	bArm1HorzULD1Unhook_00 AT %MX20356.0 : BOOL;
	bArm1HorzULD1Unhook_01 AT %MX20356.1 : BOOL;
	bArm1HorzULD1Unhook_02 AT %MX20356.2 : BOOL;
	bArm1HorzULD1Unhook_03 AT %MX20356.3 : BOOL;
	bArm1HorzULD1Unhook_04 AT %MX20356.4 : BOOL;
	bArm1HorzULD1Unhook_05 AT %MX20356.5 : BOOL;
	bArm1HorzULD1Unhook_06 AT %MX20356.6 : BOOL;
	bArm1HorzULD1Unhook_07 AT %MX20356.7 : BOOL;
	bArm1HorzULD1Unhook_08 AT %MX20356.8 : BOOL;
	bArm1HorzULD1Unhook_09 AT %MX20356.9 : BOOL;
	bArm1HorzULD1Unhook_10 AT %MX20356.10 : BOOL;
	bArm1HorzULD1Unhook_11 AT %MX20356.11 : BOOL;
	bArm1HorzULD1Unhook_12 AT %MX20356.12 : BOOL;
	bArm1HorzULD1Unhook_13 AT %MX20356.13 : BOOL;
	bArm1HorzULD1Unhook_14 AT %MX20356.14 : BOOL;
	bArm1HorzULD1Unhook_15 AT %MX20356.15 : BOOL;
	bArm1HorzULD1Unhook_16 AT %MX20356.16 : BOOL;
	bArm1HorzULD1Unhook_17 AT %MX20356.17 : BOOL;
	bArm1HorzULD1Unhook_18 AT %MX20356.18 : BOOL;
	bArm1HorzULD1Unhook_19 AT %MX20356.19 : BOOL;
	bArm1HorzULD1Unhook_20 AT %MX20356.20 : BOOL;
	bArm1HorzULD1Unhook_21 AT %MX20356.21 : BOOL;
	bArm1HorzULD1Unhook_22 AT %MX20356.22 : BOOL;
	bArm1HorzULD1Unhook_23 AT %MX20356.23 : BOOL;
	bArm1HorzULD1Unhook_24 AT %MX20356.24 : BOOL;
	bArm1HorzULD1Unhook_25 AT %MX20356.25 : BOOL;
	bArm1HorzULD1Unhook_26 AT %MX20356.26 : BOOL;
	bArm1HorzULD1Unhook_27 AT %MX20356.27 : BOOL;
	bArm1HorzULD1Unhook_28 AT %MX20356.28 : BOOL;
	bArm1HorzULD1Unhook_29 AT %MX20356.29 : BOOL;
	bArm1HorzULD1Unhook_30 AT %MX20356.30 : BOOL;
	bArm1HorzULD1Unhook_31 AT %MX20356.31 : BOOL;

	bArm1HorzStn1Unhook_00 AT %MX20304.0 : BOOL;
	bArm1HorzStn1Unhook_01 AT %MX20304.1 : BOOL;
	bArm1HorzStn1Unhook_02 AT %MX20304.2 : BOOL;
	bArm1HorzStn1Unhook_03 AT %MX20304.3 : BOOL;
	bArm1HorzStn1Unhook_04 AT %MX20304.4 : BOOL;
	bArm1HorzStn1Unhook_05 AT %MX20304.5 : BOOL;
	bArm1HorzStn1Unhook_06 AT %MX20304.6 : BOOL;
	bArm1HorzStn1Unhook_07 AT %MX20304.7 : BOOL;
	bArm1HorzStn1Unhook_08 AT %MX20304.8 : BOOL;
	bArm1HorzStn1Unhook_09 AT %MX20304.9 : BOOL;
	bArm1HorzStn1Unhook_10 AT %MX20304.10 : BOOL;
	bArm1HorzStn1Unhook_11 AT %MX20304.11 : BOOL;
	bArm1HorzStn1Unhook_12 AT %MX20304.12 : BOOL;
	bArm1HorzStn1Unhook_13 AT %MX20304.13 : BOOL;
	bArm1HorzStn1Unhook_14 AT %MX20304.14 : BOOL;
	bArm1HorzStn1Unhook_15 AT %MX20304.15 : BOOL;
	bArm1HorzStn1Unhook_16 AT %MX20304.16 : BOOL;
	bArm1HorzStn1Unhook_17 AT %MX20304.17 : BOOL;
	bArm1HorzStn1Unhook_18 AT %MX20304.18 : BOOL;
	bArm1HorzStn1Unhook_19 AT %MX20304.19 : BOOL;
	bArm1HorzStn1Unhook_20 AT %MX20304.20 : BOOL;
	bArm1HorzStn1Unhook_21 AT %MX20304.21 : BOOL;
	bArm1HorzStn1Unhook_22 AT %MX20304.22 : BOOL;
	bArm1HorzStn1Unhook_23 AT %MX20304.23 : BOOL;
	bArm1HorzStn1Unhook_24 AT %MX20304.24 : BOOL;
	bArm1HorzStn1Unhook_25 AT %MX20304.25 : BOOL;
	bArm1HorzStn1Unhook_26 AT %MX20304.26 : BOOL;
	bArm1HorzStn1Unhook_27 AT %MX20304.27 : BOOL;
	bArm1HorzStn1Unhook_28 AT %MX20304.28 : BOOL;
	bArm1HorzStn1Unhook_29 AT %MX20304.29 : BOOL;
	bArm1HorzStn1Unhook_30 AT %MX20304.30 : BOOL;
	bArm1HorzStn1Unhook_31 AT %MX20304.31 : BOOL;

	bArm1HorzStn2Unhook_00 AT %MX20308.0 : BOOL;
	bArm1HorzStn2Unhook_01 AT %MX20308.1 : BOOL;
	bArm1HorzStn2Unhook_02 AT %MX20308.2 : BOOL;
	bArm1HorzStn2Unhook_03 AT %MX20308.3 : BOOL;
	bArm1HorzStn2Unhook_04 AT %MX20308.4 : BOOL;
	bArm1HorzStn2Unhook_05 AT %MX20308.5 : BOOL;
	bArm1HorzStn2Unhook_06 AT %MX20308.6 : BOOL;
	bArm1HorzStn2Unhook_07 AT %MX20308.7 : BOOL;
	bArm1HorzStn2Unhook_08 AT %MX20308.8 : BOOL;
	bArm1HorzStn2Unhook_09 AT %MX20308.9 : BOOL;
	bArm1HorzStn2Unhook_10 AT %MX20308.10 : BOOL;
	bArm1HorzStn2Unhook_11 AT %MX20308.11 : BOOL;
	bArm1HorzStn2Unhook_12 AT %MX20308.12 : BOOL;
	bArm1HorzStn2Unhook_13 AT %MX20308.13 : BOOL;
	bArm1HorzStn2Unhook_14 AT %MX20308.14 : BOOL;
	bArm1HorzStn2Unhook_15 AT %MX20308.15 : BOOL;
	bArm1HorzStn2Unhook_16 AT %MX20308.16 : BOOL;
	bArm1HorzStn2Unhook_17 AT %MX20308.17 : BOOL;
	bArm1HorzStn2Unhook_18 AT %MX20308.18 : BOOL;
	bArm1HorzStn2Unhook_19 AT %MX20308.19 : BOOL;
	bArm1HorzStn2Unhook_20 AT %MX20308.20 : BOOL;
	bArm1HorzStn2Unhook_21 AT %MX20308.21 : BOOL;
	bArm1HorzStn2Unhook_22 AT %MX20308.22 : BOOL;
	bArm1HorzStn2Unhook_23 AT %MX20308.23 : BOOL;
	bArm1HorzStn2Unhook_24 AT %MX20308.24 : BOOL;
	bArm1HorzStn2Unhook_25 AT %MX20308.25 : BOOL;
	bArm1HorzStn2Unhook_26 AT %MX20308.26 : BOOL;
	bArm1HorzStn2Unhook_27 AT %MX20308.27 : BOOL;
	bArm1HorzStn2Unhook_28 AT %MX20308.28 : BOOL;
	bArm1HorzStn2Unhook_29 AT %MX20308.29 : BOOL;
	bArm1HorzStn2Unhook_30 AT %MX20308.30 : BOOL;
	bArm1HorzStn2Unhook_31 AT %MX20308.31 : BOOL;

	bArm1HorzStn3Unhook_00 AT %MX20312.0 : BOOL;
	bArm1HorzStn3Unhook_01 AT %MX20312.1 : BOOL;
	bArm1HorzStn3Unhook_02 AT %MX20312.2 : BOOL;
	bArm1HorzStn3Unhook_03 AT %MX20312.3 : BOOL;
	bArm1HorzStn3Unhook_04 AT %MX20312.4 : BOOL;
	bArm1HorzStn3Unhook_05 AT %MX20312.5 : BOOL;
	bArm1HorzStn3Unhook_06 AT %MX20312.6 : BOOL;
	bArm1HorzStn3Unhook_07 AT %MX20312.7 : BOOL;
	bArm1HorzStn3Unhook_08 AT %MX20312.8 : BOOL;
	bArm1HorzStn3Unhook_09 AT %MX20312.9 : BOOL;
	bArm1HorzStn3Unhook_10 AT %MX20312.10 : BOOL;
	bArm1HorzStn3Unhook_11 AT %MX20312.11 : BOOL;
	bArm1HorzStn3Unhook_12 AT %MX20312.12 : BOOL;
	bArm1HorzStn3Unhook_13 AT %MX20312.13 : BOOL;
	bArm1HorzStn3Unhook_14 AT %MX20312.14 : BOOL;
	bArm1HorzStn3Unhook_15 AT %MX20312.15 : BOOL;
	bArm1HorzStn3Unhook_16 AT %MX20312.16 : BOOL;
	bArm1HorzStn3Unhook_17 AT %MX20312.17 : BOOL;
	bArm1HorzStn3Unhook_18 AT %MX20312.18 : BOOL;
	bArm1HorzStn3Unhook_19 AT %MX20312.19 : BOOL;
	bArm1HorzStn3Unhook_20 AT %MX20312.20 : BOOL;
	bArm1HorzStn3Unhook_21 AT %MX20312.21 : BOOL;
	bArm1HorzStn3Unhook_22 AT %MX20312.22 : BOOL;
	bArm1HorzStn3Unhook_23 AT %MX20312.23 : BOOL;
	bArm1HorzStn3Unhook_24 AT %MX20312.24 : BOOL;
	bArm1HorzStn3Unhook_25 AT %MX20312.25 : BOOL;
	bArm1HorzStn3Unhook_26 AT %MX20312.26 : BOOL;
	bArm1HorzStn3Unhook_27 AT %MX20312.27 : BOOL;
	bArm1HorzStn3Unhook_28 AT %MX20312.28 : BOOL;
	bArm1HorzStn3Unhook_29 AT %MX20312.29 : BOOL;
	bArm1HorzStn3Unhook_30 AT %MX20312.30 : BOOL;
	bArm1HorzStn3Unhook_31 AT %MX20312.31 : BOOL;

	bArm1HorzStn4Unhook_00 AT %MX20316.0 : BOOL;
	bArm1HorzStn4Unhook_01 AT %MX20316.1 : BOOL;
	bArm1HorzStn4Unhook_02 AT %MX20316.2 : BOOL;
	bArm1HorzStn4Unhook_03 AT %MX20316.3 : BOOL;
	bArm1HorzStn4Unhook_04 AT %MX20316.4 : BOOL;
	bArm1HorzStn4Unhook_05 AT %MX20316.5 : BOOL;
	bArm1HorzStn4Unhook_06 AT %MX20316.6 : BOOL;
	bArm1HorzStn4Unhook_07 AT %MX20316.7 : BOOL;
	bArm1HorzStn4Unhook_08 AT %MX20316.8 : BOOL;
	bArm1HorzStn4Unhook_09 AT %MX20316.9 : BOOL;
	bArm1HorzStn4Unhook_10 AT %MX20316.10 : BOOL;
	bArm1HorzStn4Unhook_11 AT %MX20316.11 : BOOL;
	bArm1HorzStn4Unhook_12 AT %MX20316.12 : BOOL;
	bArm1HorzStn4Unhook_13 AT %MX20316.13 : BOOL;
	bArm1HorzStn4Unhook_14 AT %MX20316.14 : BOOL;
	bArm1HorzStn4Unhook_15 AT %MX20316.15 : BOOL;
	bArm1HorzStn4Unhook_16 AT %MX20316.16 : BOOL;
	bArm1HorzStn4Unhook_17 AT %MX20316.17 : BOOL;
	bArm1HorzStn4Unhook_18 AT %MX20316.18 : BOOL;
	bArm1HorzStn4Unhook_19 AT %MX20316.19 : BOOL;
	bArm1HorzStn4Unhook_20 AT %MX20316.20 : BOOL;
	bArm1HorzStn4Unhook_21 AT %MX20316.21 : BOOL;
	bArm1HorzStn4Unhook_22 AT %MX20316.22 : BOOL;
	bArm1HorzStn4Unhook_23 AT %MX20316.23 : BOOL;
	bArm1HorzStn4Unhook_24 AT %MX20316.24 : BOOL;
	bArm1HorzStn4Unhook_25 AT %MX20316.25 : BOOL;
	bArm1HorzStn4Unhook_26 AT %MX20316.26 : BOOL;
	bArm1HorzStn4Unhook_27 AT %MX20316.27 : BOOL;
	bArm1HorzStn4Unhook_28 AT %MX20316.28 : BOOL;
	bArm1HorzStn4Unhook_29 AT %MX20316.29 : BOOL;
	bArm1HorzStn4Unhook_30 AT %MX20316.30 : BOOL;
	bArm1HorzStn4Unhook_31 AT %MX20316.31 : BOOL;

	bArm1HorzStn5Unhook_00 AT %MX20320.0 : BOOL;
	bArm1HorzStn5Unhook_01 AT %MX20320.1 : BOOL;
	bArm1HorzStn5Unhook_02 AT %MX20320.2 : BOOL;
	bArm1HorzStn5Unhook_03 AT %MX20320.3 : BOOL;
	bArm1HorzStn5Unhook_04 AT %MX20320.4 : BOOL;
	bArm1HorzStn5Unhook_05 AT %MX20320.5 : BOOL;
	bArm1HorzStn5Unhook_06 AT %MX20320.6 : BOOL;
	bArm1HorzStn5Unhook_07 AT %MX20320.7 : BOOL;
	bArm1HorzStn5Unhook_08 AT %MX20320.8 : BOOL;
	bArm1HorzStn5Unhook_09 AT %MX20320.9 : BOOL;
	bArm1HorzStn5Unhook_10 AT %MX20320.10 : BOOL;
	bArm1HorzStn5Unhook_11 AT %MX20320.11 : BOOL;
	bArm1HorzStn5Unhook_12 AT %MX20320.12 : BOOL;
	bArm1HorzStn5Unhook_13 AT %MX20320.13 : BOOL;
	bArm1HorzStn5Unhook_14 AT %MX20320.14 : BOOL;
	bArm1HorzStn5Unhook_15 AT %MX20320.15 : BOOL;
	bArm1HorzStn5Unhook_16 AT %MX20320.16 : BOOL;
	bArm1HorzStn5Unhook_17 AT %MX20320.17 : BOOL;
	bArm1HorzStn5Unhook_18 AT %MX20320.18 : BOOL;
	bArm1HorzStn5Unhook_19 AT %MX20320.19 : BOOL;
	bArm1HorzStn5Unhook_20 AT %MX20320.20 : BOOL;
	bArm1HorzStn5Unhook_21 AT %MX20320.21 : BOOL;
	bArm1HorzStn5Unhook_22 AT %MX20320.22 : BOOL;
	bArm1HorzStn5Unhook_23 AT %MX20320.23 : BOOL;
	bArm1HorzStn5Unhook_24 AT %MX20320.24 : BOOL;
	bArm1HorzStn5Unhook_25 AT %MX20320.25 : BOOL;
	bArm1HorzStn5Unhook_26 AT %MX20320.26 : BOOL;
	bArm1HorzStn5Unhook_27 AT %MX20320.27 : BOOL;
	bArm1HorzStn5Unhook_28 AT %MX20320.28 : BOOL;
	bArm1HorzStn5Unhook_29 AT %MX20320.29 : BOOL;
	bArm1HorzStn5Unhook_30 AT %MX20320.30 : BOOL;
	bArm1HorzStn5Unhook_31 AT %MX20320.31 : BOOL;

	bArm1HorzStn6Unhook_00 AT %MX20324.0 : BOOL;
	bArm1HorzStn6Unhook_01 AT %MX20324.1 : BOOL;
	bArm1HorzStn6Unhook_02 AT %MX20324.2 : BOOL;
	bArm1HorzStn6Unhook_03 AT %MX20324.3 : BOOL;
	bArm1HorzStn6Unhook_04 AT %MX20324.4 : BOOL;
	bArm1HorzStn6Unhook_05 AT %MX20324.5 : BOOL;
	bArm1HorzStn6Unhook_06 AT %MX20324.6 : BOOL;
	bArm1HorzStn6Unhook_07 AT %MX20324.7 : BOOL;
	bArm1HorzStn6Unhook_08 AT %MX20324.8 : BOOL;
	bArm1HorzStn6Unhook_09 AT %MX20324.9 : BOOL;
	bArm1HorzStn6Unhook_10 AT %MX20324.10 : BOOL;
	bArm1HorzStn6Unhook_11 AT %MX20324.11 : BOOL;
	bArm1HorzStn6Unhook_12 AT %MX20324.12 : BOOL;
	bArm1HorzStn6Unhook_13 AT %MX20324.13 : BOOL;
	bArm1HorzStn6Unhook_14 AT %MX20324.14 : BOOL;
	bArm1HorzStn6Unhook_15 AT %MX20324.15 : BOOL;
	bArm1HorzStn6Unhook_16 AT %MX20324.16 : BOOL;
	bArm1HorzStn6Unhook_17 AT %MX20324.17 : BOOL;
	bArm1HorzStn6Unhook_18 AT %MX20324.18 : BOOL;
	bArm1HorzStn6Unhook_19 AT %MX20324.19 : BOOL;
	bArm1HorzStn6Unhook_20 AT %MX20324.20 : BOOL;
	bArm1HorzStn6Unhook_21 AT %MX20324.21 : BOOL;
	bArm1HorzStn6Unhook_22 AT %MX20324.22 : BOOL;
	bArm1HorzStn6Unhook_23 AT %MX20324.23 : BOOL;
	bArm1HorzStn6Unhook_24 AT %MX20324.24 : BOOL;
	bArm1HorzStn6Unhook_25 AT %MX20324.25 : BOOL;
	bArm1HorzStn6Unhook_26 AT %MX20324.26 : BOOL;
	bArm1HorzStn6Unhook_27 AT %MX20324.27 : BOOL;
	bArm1HorzStn6Unhook_28 AT %MX20324.28 : BOOL;
	bArm1HorzStn6Unhook_29 AT %MX20324.29 : BOOL;
	bArm1HorzStn6Unhook_30 AT %MX20324.30 : BOOL;
	bArm1HorzStn6Unhook_31 AT %MX20324.31 : BOOL;

	bArm1HorzStn7Unhook_00 AT %MX20328.0 : BOOL;
	bArm1HorzStn7Unhook_01 AT %MX20328.1 : BOOL;
	bArm1HorzStn7Unhook_02 AT %MX20328.2 : BOOL;
	bArm1HorzStn7Unhook_03 AT %MX20328.3 : BOOL;
	bArm1HorzStn7Unhook_04 AT %MX20328.4 : BOOL;
	bArm1HorzStn7Unhook_05 AT %MX20328.5 : BOOL;
	bArm1HorzStn7Unhook_06 AT %MX20328.6 : BOOL;
	bArm1HorzStn7Unhook_07 AT %MX20328.7 : BOOL;
	bArm1HorzStn7Unhook_08 AT %MX20328.8 : BOOL;
	bArm1HorzStn7Unhook_09 AT %MX20328.9 : BOOL;
	bArm1HorzStn7Unhook_10 AT %MX20328.10 : BOOL;
	bArm1HorzStn7Unhook_11 AT %MX20328.11 : BOOL;
	bArm1HorzStn7Unhook_12 AT %MX20328.12 : BOOL;
	bArm1HorzStn7Unhook_13 AT %MX20328.13 : BOOL;
	bArm1HorzStn7Unhook_14 AT %MX20328.14 : BOOL;
	bArm1HorzStn7Unhook_15 AT %MX20328.15 : BOOL;
	bArm1HorzStn7Unhook_16 AT %MX20328.16 : BOOL;
	bArm1HorzStn7Unhook_17 AT %MX20328.17 : BOOL;
	bArm1HorzStn7Unhook_18 AT %MX20328.18 : BOOL;
	bArm1HorzStn7Unhook_19 AT %MX20328.19 : BOOL;
	bArm1HorzStn7Unhook_20 AT %MX20328.20 : BOOL;
	bArm1HorzStn7Unhook_21 AT %MX20328.21 : BOOL;
	bArm1HorzStn7Unhook_22 AT %MX20328.22 : BOOL;
	bArm1HorzStn7Unhook_23 AT %MX20328.23 : BOOL;
	bArm1HorzStn7Unhook_24 AT %MX20328.24 : BOOL;
	bArm1HorzStn7Unhook_25 AT %MX20328.25 : BOOL;
	bArm1HorzStn7Unhook_26 AT %MX20328.26 : BOOL;
	bArm1HorzStn7Unhook_27 AT %MX20328.27 : BOOL;
	bArm1HorzStn7Unhook_28 AT %MX20328.28 : BOOL;
	bArm1HorzStn7Unhook_29 AT %MX20328.29 : BOOL;
	bArm1HorzStn7Unhook_30 AT %MX20328.30 : BOOL;
	bArm1HorzStn7Unhook_31 AT %MX20328.31 : BOOL;

	bArm1HorzStn8Unhook_00 AT %MX20332.0 : BOOL;
	bArm1HorzStn8Unhook_01 AT %MX20332.1 : BOOL;
	bArm1HorzStn8Unhook_02 AT %MX20332.2 : BOOL;
	bArm1HorzStn8Unhook_03 AT %MX20332.3 : BOOL;
	bArm1HorzStn8Unhook_04 AT %MX20332.4 : BOOL;
	bArm1HorzStn8Unhook_05 AT %MX20332.5 : BOOL;
	bArm1HorzStn8Unhook_06 AT %MX20332.6 : BOOL;
	bArm1HorzStn8Unhook_07 AT %MX20332.7 : BOOL;
	bArm1HorzStn8Unhook_08 AT %MX20332.8 : BOOL;
	bArm1HorzStn8Unhook_09 AT %MX20332.9 : BOOL;
	bArm1HorzStn8Unhook_10 AT %MX20332.10 : BOOL;
	bArm1HorzStn8Unhook_11 AT %MX20332.11 : BOOL;
	bArm1HorzStn8Unhook_12 AT %MX20332.12 : BOOL;
	bArm1HorzStn8Unhook_13 AT %MX20332.13 : BOOL;
	bArm1HorzStn8Unhook_14 AT %MX20332.14 : BOOL;
	bArm1HorzStn8Unhook_15 AT %MX20332.15 : BOOL;
	bArm1HorzStn8Unhook_16 AT %MX20332.16 : BOOL;
	bArm1HorzStn8Unhook_17 AT %MX20332.17 : BOOL;
	bArm1HorzStn8Unhook_18 AT %MX20332.18 : BOOL;
	bArm1HorzStn8Unhook_19 AT %MX20332.19 : BOOL;
	bArm1HorzStn8Unhook_20 AT %MX20332.20 : BOOL;
	bArm1HorzStn8Unhook_21 AT %MX20332.21 : BOOL;
	bArm1HorzStn8Unhook_22 AT %MX20332.22 : BOOL;
	bArm1HorzStn8Unhook_23 AT %MX20332.23 : BOOL;
	bArm1HorzStn8Unhook_24 AT %MX20332.24 : BOOL;
	bArm1HorzStn8Unhook_25 AT %MX20332.25 : BOOL;
	bArm1HorzStn8Unhook_26 AT %MX20332.26 : BOOL;
	bArm1HorzStn8Unhook_27 AT %MX20332.27 : BOOL;
	bArm1HorzStn8Unhook_28 AT %MX20332.28 : BOOL;
	bArm1HorzStn8Unhook_29 AT %MX20332.29 : BOOL;
	bArm1HorzStn8Unhook_30 AT %MX20332.30 : BOOL;
	bArm1HorzStn8Unhook_31 AT %MX20332.31 : BOOL;

	bArm1HorzStn9Unhook_00 AT %MX20336.0 : BOOL;
	bArm1HorzStn9Unhook_01 AT %MX20336.1 : BOOL;
	bArm1HorzStn9Unhook_02 AT %MX20336.2 : BOOL;
	bArm1HorzStn9Unhook_03 AT %MX20336.3 : BOOL;
	bArm1HorzStn9Unhook_04 AT %MX20336.4 : BOOL;
	bArm1HorzStn9Unhook_05 AT %MX20336.5 : BOOL;
	bArm1HorzStn9Unhook_06 AT %MX20336.6 : BOOL;
	bArm1HorzStn9Unhook_07 AT %MX20336.7 : BOOL;
	bArm1HorzStn9Unhook_08 AT %MX20336.8 : BOOL;
	bArm1HorzStn9Unhook_09 AT %MX20336.9 : BOOL;
	bArm1HorzStn9Unhook_10 AT %MX20336.10 : BOOL;
	bArm1HorzStn9Unhook_11 AT %MX20336.11 : BOOL;
	bArm1HorzStn9Unhook_12 AT %MX20336.12 : BOOL;
	bArm1HorzStn9Unhook_13 AT %MX20336.13 : BOOL;
	bArm1HorzStn9Unhook_14 AT %MX20336.14 : BOOL;
	bArm1HorzStn9Unhook_15 AT %MX20336.15 : BOOL;
	bArm1HorzStn9Unhook_16 AT %MX20336.16 : BOOL;
	bArm1HorzStn9Unhook_17 AT %MX20336.17 : BOOL;
	bArm1HorzStn9Unhook_18 AT %MX20336.18 : BOOL;
	bArm1HorzStn9Unhook_19 AT %MX20336.19 : BOOL;
	bArm1HorzStn9Unhook_20 AT %MX20336.20 : BOOL;
	bArm1HorzStn9Unhook_21 AT %MX20336.21 : BOOL;
	bArm1HorzStn9Unhook_22 AT %MX20336.22 : BOOL;
	bArm1HorzStn9Unhook_23 AT %MX20336.23 : BOOL;
	bArm1HorzStn9Unhook_24 AT %MX20336.24 : BOOL;
	bArm1HorzStn9Unhook_25 AT %MX20336.25 : BOOL;
	bArm1HorzStn9Unhook_26 AT %MX20336.26 : BOOL;
	bArm1HorzStn9Unhook_27 AT %MX20336.27 : BOOL;
	bArm1HorzStn9Unhook_28 AT %MX20336.28 : BOOL;
	bArm1HorzStn9Unhook_29 AT %MX20336.29 : BOOL;
	bArm1HorzStn9Unhook_30 AT %MX20336.30 : BOOL;
	bArm1HorzStn9Unhook_31 AT %MX20336.31 : BOOL;

	bArm1HorzStn10Unhook_00 AT %MX20340.0 : BOOL;
	bArm1HorzStn10Unhook_01 AT %MX20340.1 : BOOL;
	bArm1HorzStn10Unhook_02 AT %MX20340.2 : BOOL;
	bArm1HorzStn10Unhook_03 AT %MX20340.3 : BOOL;
	bArm1HorzStn10Unhook_04 AT %MX20340.4 : BOOL;
	bArm1HorzStn10Unhook_05 AT %MX20340.5 : BOOL;
	bArm1HorzStn10Unhook_06 AT %MX20340.6 : BOOL;
	bArm1HorzStn10Unhook_07 AT %MX20340.7 : BOOL;
	bArm1HorzStn10Unhook_08 AT %MX20340.8 : BOOL;
	bArm1HorzStn10Unhook_09 AT %MX20340.9 : BOOL;
	bArm1HorzStn10Unhook_10 AT %MX20340.10 : BOOL;
	bArm1HorzStn10Unhook_11 AT %MX20340.11 : BOOL;
	bArm1HorzStn10Unhook_12 AT %MX20340.12 : BOOL;
	bArm1HorzStn10Unhook_13 AT %MX20340.13 : BOOL;
	bArm1HorzStn10Unhook_14 AT %MX20340.14 : BOOL;
	bArm1HorzStn10Unhook_15 AT %MX20340.15 : BOOL;
	bArm1HorzStn10Unhook_16 AT %MX20340.16 : BOOL;
	bArm1HorzStn10Unhook_17 AT %MX20340.17 : BOOL;
	bArm1HorzStn10Unhook_18 AT %MX20340.18 : BOOL;
	bArm1HorzStn10Unhook_19 AT %MX20340.19 : BOOL;
	bArm1HorzStn10Unhook_20 AT %MX20340.20 : BOOL;
	bArm1HorzStn10Unhook_21 AT %MX20340.21 : BOOL;
	bArm1HorzStn10Unhook_22 AT %MX20340.22 : BOOL;
	bArm1HorzStn10Unhook_23 AT %MX20340.23 : BOOL;
	bArm1HorzStn10Unhook_24 AT %MX20340.24 : BOOL;
	bArm1HorzStn10Unhook_25 AT %MX20340.25 : BOOL;
	bArm1HorzStn10Unhook_26 AT %MX20340.26 : BOOL;
	bArm1HorzStn10Unhook_27 AT %MX20340.27 : BOOL;
	bArm1HorzStn10Unhook_28 AT %MX20340.28 : BOOL;
	bArm1HorzStn10Unhook_29 AT %MX20340.29 : BOOL;
	bArm1HorzStn10Unhook_30 AT %MX20340.30 : BOOL;
	bArm1HorzStn10Unhook_31 AT %MX20340.31 : BOOL;

	bArm1HorzStn11Unhook_00 AT %MX20344.0 : BOOL;
	bArm1HorzStn11Unhook_01 AT %MX20344.1 : BOOL;
	bArm1HorzStn11Unhook_02 AT %MX20344.2 : BOOL;
	bArm1HorzStn11Unhook_03 AT %MX20344.3 : BOOL;
	bArm1HorzStn11Unhook_04 AT %MX20344.4 : BOOL;
	bArm1HorzStn11Unhook_05 AT %MX20344.5 : BOOL;
	bArm1HorzStn11Unhook_06 AT %MX20344.6 : BOOL;
	bArm1HorzStn11Unhook_07 AT %MX20344.7 : BOOL;
	bArm1HorzStn11Unhook_08 AT %MX20344.8 : BOOL;
	bArm1HorzStn11Unhook_09 AT %MX20344.9 : BOOL;
	bArm1HorzStn11Unhook_10 AT %MX20344.10 : BOOL;
	bArm1HorzStn11Unhook_11 AT %MX20344.11 : BOOL;
	bArm1HorzStn11Unhook_12 AT %MX20344.12 : BOOL;
	bArm1HorzStn11Unhook_13 AT %MX20344.13 : BOOL;
	bArm1HorzStn11Unhook_14 AT %MX20344.14 : BOOL;
	bArm1HorzStn11Unhook_15 AT %MX20344.15 : BOOL;
	bArm1HorzStn11Unhook_16 AT %MX20344.16 : BOOL;
	bArm1HorzStn11Unhook_17 AT %MX20344.17 : BOOL;
	bArm1HorzStn11Unhook_18 AT %MX20344.18 : BOOL;
	bArm1HorzStn11Unhook_19 AT %MX20344.19 : BOOL;
	bArm1HorzStn11Unhook_20 AT %MX20344.20 : BOOL;
	bArm1HorzStn11Unhook_21 AT %MX20344.21 : BOOL;
	bArm1HorzStn11Unhook_22 AT %MX20344.22 : BOOL;
	bArm1HorzStn11Unhook_23 AT %MX20344.23 : BOOL;
	bArm1HorzStn11Unhook_24 AT %MX20344.24 : BOOL;
	bArm1HorzStn11Unhook_25 AT %MX20344.25 : BOOL;
	bArm1HorzStn11Unhook_26 AT %MX20344.26 : BOOL;
	bArm1HorzStn11Unhook_27 AT %MX20344.27 : BOOL;
	bArm1HorzStn11Unhook_28 AT %MX20344.28 : BOOL;
	bArm1HorzStn11Unhook_29 AT %MX20344.29 : BOOL;
	bArm1HorzStn11Unhook_30 AT %MX20344.30 : BOOL;
	bArm1HorzStn11Unhook_31 AT %MX20344.31 : BOOL;

	bArm1HorzStn12Unhook_00 AT %MX20348.0 : BOOL;
	bArm1HorzStn12Unhook_01 AT %MX20348.1 : BOOL;
	bArm1HorzStn12Unhook_02 AT %MX20348.2 : BOOL;
	bArm1HorzStn12Unhook_03 AT %MX20348.3 : BOOL;
	bArm1HorzStn12Unhook_04 AT %MX20348.4 : BOOL;
	bArm1HorzStn12Unhook_05 AT %MX20348.5 : BOOL;
	bArm1HorzStn12Unhook_06 AT %MX20348.6 : BOOL;
	bArm1HorzStn12Unhook_07 AT %MX20348.7 : BOOL;
	bArm1HorzStn12Unhook_08 AT %MX20348.8 : BOOL;
	bArm1HorzStn12Unhook_09 AT %MX20348.9 : BOOL;
	bArm1HorzStn12Unhook_10 AT %MX20348.10 : BOOL;
	bArm1HorzStn12Unhook_11 AT %MX20348.11 : BOOL;
	bArm1HorzStn12Unhook_12 AT %MX20348.12 : BOOL;
	bArm1HorzStn12Unhook_13 AT %MX20348.13 : BOOL;
	bArm1HorzStn12Unhook_14 AT %MX20348.14 : BOOL;
	bArm1HorzStn12Unhook_15 AT %MX20348.15 : BOOL;
	bArm1HorzStn12Unhook_16 AT %MX20348.16 : BOOL;
	bArm1HorzStn12Unhook_17 AT %MX20348.17 : BOOL;
	bArm1HorzStn12Unhook_18 AT %MX20348.18 : BOOL;
	bArm1HorzStn12Unhook_19 AT %MX20348.19 : BOOL;
	bArm1HorzStn12Unhook_20 AT %MX20348.20 : BOOL;
	bArm1HorzStn12Unhook_21 AT %MX20348.21 : BOOL;
	bArm1HorzStn12Unhook_22 AT %MX20348.22 : BOOL;
	bArm1HorzStn12Unhook_23 AT %MX20348.23 : BOOL;
	bArm1HorzStn12Unhook_24 AT %MX20348.24 : BOOL;
	bArm1HorzStn12Unhook_25 AT %MX20348.25 : BOOL;
	bArm1HorzStn12Unhook_26 AT %MX20348.26 : BOOL;
	bArm1HorzStn12Unhook_27 AT %MX20348.27 : BOOL;
	bArm1HorzStn12Unhook_28 AT %MX20348.28 : BOOL;
	bArm1HorzStn12Unhook_29 AT %MX20348.29 : BOOL;
	bArm1HorzStn12Unhook_30 AT %MX20348.30 : BOOL;
	bArm1HorzStn12Unhook_31 AT %MX20348.31 : BOOL;


(* xxxxxxxxxxxxxxxxxxxxxxxxxxxxxxxxxxxxxxx Vert xxxxxxxxxxxxxxxxxxxxxxxxxxxxxxxxxxxxxxx*)
(*========= Up BOOL LINK with %MX25000-MX25099 =========*)

	bArm1VertLD1Up_00 AT %MX25052.0 : BOOL;
	bArm1VertLD1Up_01 AT %MX25052.1 : BOOL;
	bArm1VertLD1Up_02 AT %MX25052.2 : BOOL;
	bArm1VertLD1Up_03 AT %MX25052.3 : BOOL;
	bArm1VertLD1Up_04 AT %MX25052.4 : BOOL;
	bArm1VertLD1Up_05 AT %MX25052.5 : BOOL;
	bArm1VertLD1Up_06 AT %MX25052.6 : BOOL;
	bArm1VertLD1Up_07 AT %MX25052.7 : BOOL;
	bArm1VertLD1Up_08 AT %MX25052.8 : BOOL;
	bArm1VertLD1Up_09 AT %MX25052.9 : BOOL;
	bArm1VertLD1Up_10 AT %MX25052.10 : BOOL;
	bArm1VertLD1Up_11 AT %MX25052.11 : BOOL;
	bArm1VertLD1Up_12 AT %MX25052.12 : BOOL;
	bArm1VertLD1Up_13 AT %MX25052.13 : BOOL;
	bArm1VertLD1Up_14 AT %MX25052.14 : BOOL;
	bArm1VertLD1Up_15 AT %MX25052.15 : BOOL;
	bArm1VertLD1Up_16 AT %MX25052.16 : BOOL;
	bArm1VertLD1Up_17 AT %MX25052.17 : BOOL;
	bArm1VertLD1Up_18 AT %MX25052.18 : BOOL;
	bArm1VertLD1Up_19 AT %MX25052.19 : BOOL;
	bArm1VertLD1Up_20 AT %MX25052.20 : BOOL;
	bArm1VertLD1Up_21 AT %MX25052.21 : BOOL;
	bArm1VertLD1Up_22 AT %MX25052.22 : BOOL;
	bArm1VertLD1Up_23 AT %MX25052.23 : BOOL;
	bArm1VertLD1Up_24 AT %MX25052.24 : BOOL;
	bArm1VertLD1Up_25 AT %MX25052.25 : BOOL;
	bArm1VertLD1Up_26 AT %MX25052.26 : BOOL;
	bArm1VertLD1Up_27 AT %MX25052.27 : BOOL;
	bArm1VertLD1Up_28 AT %MX25052.28 : BOOL;
	bArm1VertLD1Up_29 AT %MX25052.29 : BOOL;
	bArm1VertLD1Up_30 AT %MX25052.30 : BOOL;
	bArm1VertLD1Up_31 AT %MX25052.31 : BOOL;

	bArm1VertULD1Up_00 AT %MX25056.0 : BOOL;
	bArm1VertULD1Up_01 AT %MX25056.1 : BOOL;
	bArm1VertULD1Up_02 AT %MX25056.2 : BOOL;
	bArm1VertULD1Up_03 AT %MX25056.3 : BOOL;
	bArm1VertULD1Up_04 AT %MX25056.4 : BOOL;
	bArm1VertULD1Up_05 AT %MX25056.5 : BOOL;
	bArm1VertULD1Up_06 AT %MX25056.6 : BOOL;
	bArm1VertULD1Up_07 AT %MX25056.7 : BOOL;
	bArm1VertULD1Up_08 AT %MX25056.8 : BOOL;
	bArm1VertULD1Up_09 AT %MX25056.9 : BOOL;
	bArm1VertULD1Up_10 AT %MX25056.10 : BOOL;
	bArm1VertULD1Up_11 AT %MX25056.11 : BOOL;
	bArm1VertULD1Up_12 AT %MX25056.12 : BOOL;
	bArm1VertULD1Up_13 AT %MX25056.13 : BOOL;
	bArm1VertULD1Up_14 AT %MX25056.14 : BOOL;
	bArm1VertULD1Up_15 AT %MX25056.15 : BOOL;
	bArm1VertULD1Up_16 AT %MX25056.16 : BOOL;
	bArm1VertULD1Up_17 AT %MX25056.17 : BOOL;
	bArm1VertULD1Up_18 AT %MX25056.18 : BOOL;
	bArm1VertULD1Up_19 AT %MX25056.19 : BOOL;
	bArm1VertULD1Up_20 AT %MX25056.20 : BOOL;
	bArm1VertULD1Up_21 AT %MX25056.21 : BOOL;
	bArm1VertULD1Up_22 AT %MX25056.22 : BOOL;
	bArm1VertULD1Up_23 AT %MX25056.23 : BOOL;
	bArm1VertULD1Up_24 AT %MX25056.24 : BOOL;
	bArm1VertULD1Up_25 AT %MX25056.25 : BOOL;
	bArm1VertULD1Up_26 AT %MX25056.26 : BOOL;
	bArm1VertULD1Up_27 AT %MX25056.27 : BOOL;
	bArm1VertULD1Up_28 AT %MX25056.28 : BOOL;
	bArm1VertULD1Up_29 AT %MX25056.29 : BOOL;
	bArm1VertULD1Up_30 AT %MX25056.30 : BOOL;
	bArm1VertULD1Up_31 AT %MX25056.31 : BOOL;

	bArm1VertStn1Up_00 AT %MX25004.0 : BOOL;
	bArm1VertStn1Up_01 AT %MX25004.1 : BOOL;
	bArm1VertStn1Up_02 AT %MX25004.2 : BOOL;
	bArm1VertStn1Up_03 AT %MX25004.3 : BOOL;
	bArm1VertStn1Up_04 AT %MX25004.4 : BOOL;
	bArm1VertStn1Up_05 AT %MX25004.5 : BOOL;
	bArm1VertStn1Up_06 AT %MX25004.6 : BOOL;
	bArm1VertStn1Up_07 AT %MX25004.7 : BOOL;
	bArm1VertStn1Up_08 AT %MX25004.8 : BOOL;
	bArm1VertStn1Up_09 AT %MX25004.9 : BOOL;
	bArm1VertStn1Up_10 AT %MX25004.10 : BOOL;
	bArm1VertStn1Up_11 AT %MX25004.11 : BOOL;
	bArm1VertStn1Up_12 AT %MX25004.12 : BOOL;
	bArm1VertStn1Up_13 AT %MX25004.13 : BOOL;
	bArm1VertStn1Up_14 AT %MX25004.14 : BOOL;
	bArm1VertStn1Up_15 AT %MX25004.15 : BOOL;
	bArm1VertStn1Up_16 AT %MX25004.16 : BOOL;
	bArm1VertStn1Up_17 AT %MX25004.17 : BOOL;
	bArm1VertStn1Up_18 AT %MX25004.18 : BOOL;
	bArm1VertStn1Up_19 AT %MX25004.19 : BOOL;
	bArm1VertStn1Up_20 AT %MX25004.20 : BOOL;
	bArm1VertStn1Up_21 AT %MX25004.21 : BOOL;
	bArm1VertStn1Up_22 AT %MX25004.22 : BOOL;
	bArm1VertStn1Up_23 AT %MX25004.23 : BOOL;
	bArm1VertStn1Up_24 AT %MX25004.24 : BOOL;
	bArm1VertStn1Up_25 AT %MX25004.25 : BOOL;
	bArm1VertStn1Up_26 AT %MX25004.26 : BOOL;
	bArm1VertStn1Up_27 AT %MX25004.27 : BOOL;
	bArm1VertStn1Up_28 AT %MX25004.28 : BOOL;
	bArm1VertStn1Up_29 AT %MX25004.29 : BOOL;
	bArm1VertStn1Up_30 AT %MX25004.30 : BOOL;
	bArm1VertStn1Up_31 AT %MX25004.31 : BOOL;

	bArm1VertStn2Up_00 AT %MX25008.0 : BOOL;
	bArm1VertStn2Up_01 AT %MX25008.1 : BOOL;
	bArm1VertStn2Up_02 AT %MX25008.2 : BOOL;
	bArm1VertStn2Up_03 AT %MX25008.3 : BOOL;
	bArm1VertStn2Up_04 AT %MX25008.4 : BOOL;
	bArm1VertStn2Up_05 AT %MX25008.5 : BOOL;
	bArm1VertStn2Up_06 AT %MX25008.6 : BOOL;
	bArm1VertStn2Up_07 AT %MX25008.7 : BOOL;
	bArm1VertStn2Up_08 AT %MX25008.8 : BOOL;
	bArm1VertStn2Up_09 AT %MX25008.9 : BOOL;
	bArm1VertStn2Up_10 AT %MX25008.10 : BOOL;
	bArm1VertStn2Up_11 AT %MX25008.11 : BOOL;
	bArm1VertStn2Up_12 AT %MX25008.12 : BOOL;
	bArm1VertStn2Up_13 AT %MX25008.13 : BOOL;
	bArm1VertStn2Up_14 AT %MX25008.14 : BOOL;
	bArm1VertStn2Up_15 AT %MX25008.15 : BOOL;
	bArm1VertStn2Up_16 AT %MX25008.16 : BOOL;
	bArm1VertStn2Up_17 AT %MX25008.17 : BOOL;
	bArm1VertStn2Up_18 AT %MX25008.18 : BOOL;
	bArm1VertStn2Up_19 AT %MX25008.19 : BOOL;
	bArm1VertStn2Up_20 AT %MX25008.20 : BOOL;
	bArm1VertStn2Up_21 AT %MX25008.21 : BOOL;
	bArm1VertStn2Up_22 AT %MX25008.22 : BOOL;
	bArm1VertStn2Up_23 AT %MX25008.23 : BOOL;
	bArm1VertStn2Up_24 AT %MX25008.24 : BOOL;
	bArm1VertStn2Up_25 AT %MX25008.25 : BOOL;
	bArm1VertStn2Up_26 AT %MX25008.26 : BOOL;
	bArm1VertStn2Up_27 AT %MX25008.27 : BOOL;
	bArm1VertStn2Up_28 AT %MX25008.28 : BOOL;
	bArm1VertStn2Up_29 AT %MX25008.29 : BOOL;
	bArm1VertStn2Up_30 AT %MX25008.30 : BOOL;
	bArm1VertStn2Up_31 AT %MX25008.31 : BOOL;

	bArm1VertStn3Up_00 AT %MX25012.0 : BOOL;
	bArm1VertStn3Up_01 AT %MX25012.1 : BOOL;
	bArm1VertStn3Up_02 AT %MX25012.2 : BOOL;
	bArm1VertStn3Up_03 AT %MX25012.3 : BOOL;
	bArm1VertStn3Up_04 AT %MX25012.4 : BOOL;
	bArm1VertStn3Up_05 AT %MX25012.5 : BOOL;
	bArm1VertStn3Up_06 AT %MX25012.6 : BOOL;
	bArm1VertStn3Up_07 AT %MX25012.7 : BOOL;
	bArm1VertStn3Up_08 AT %MX25012.8 : BOOL;
	bArm1VertStn3Up_09 AT %MX25012.9 : BOOL;
	bArm1VertStn3Up_10 AT %MX25012.10 : BOOL;
	bArm1VertStn3Up_11 AT %MX25012.11 : BOOL;
	bArm1VertStn3Up_12 AT %MX25012.12 : BOOL;
	bArm1VertStn3Up_13 AT %MX25012.13 : BOOL;
	bArm1VertStn3Up_14 AT %MX25012.14 : BOOL;
	bArm1VertStn3Up_15 AT %MX25012.15 : BOOL;
	bArm1VertStn3Up_16 AT %MX25012.16 : BOOL;
	bArm1VertStn3Up_17 AT %MX25012.17 : BOOL;
	bArm1VertStn3Up_18 AT %MX25012.18 : BOOL;
	bArm1VertStn3Up_19 AT %MX25012.19 : BOOL;
	bArm1VertStn3Up_20 AT %MX25012.20 : BOOL;
	bArm1VertStn3Up_21 AT %MX25012.21 : BOOL;
	bArm1VertStn3Up_22 AT %MX25012.22 : BOOL;
	bArm1VertStn3Up_23 AT %MX25012.23 : BOOL;
	bArm1VertStn3Up_24 AT %MX25012.24 : BOOL;
	bArm1VertStn3Up_25 AT %MX25012.25 : BOOL;
	bArm1VertStn3Up_26 AT %MX25012.26 : BOOL;
	bArm1VertStn3Up_27 AT %MX25012.27 : BOOL;
	bArm1VertStn3Up_28 AT %MX25012.28 : BOOL;
	bArm1VertStn3Up_29 AT %MX25012.29 : BOOL;
	bArm1VertStn3Up_30 AT %MX25012.30 : BOOL;
	bArm1VertStn3Up_31 AT %MX25012.31 : BOOL;

	bArm1VertStn4Up_00 AT %MX25016.0 : BOOL;
	bArm1VertStn4Up_01 AT %MX25016.1 : BOOL;
	bArm1VertStn4Up_02 AT %MX25016.2 : BOOL;
	bArm1VertStn4Up_03 AT %MX25016.3 : BOOL;
	bArm1VertStn4Up_04 AT %MX25016.4 : BOOL;
	bArm1VertStn4Up_05 AT %MX25016.5 : BOOL;
	bArm1VertStn4Up_06 AT %MX25016.6 : BOOL;
	bArm1VertStn4Up_07 AT %MX25016.7 : BOOL;
	bArm1VertStn4Up_08 AT %MX25016.8 : BOOL;
	bArm1VertStn4Up_09 AT %MX25016.9 : BOOL;
	bArm1VertStn4Up_10 AT %MX25016.10 : BOOL;
	bArm1VertStn4Up_11 AT %MX25016.11 : BOOL;
	bArm1VertStn4Up_12 AT %MX25016.12 : BOOL;
	bArm1VertStn4Up_13 AT %MX25016.13 : BOOL;
	bArm1VertStn4Up_14 AT %MX25016.14 : BOOL;
	bArm1VertStn4Up_15 AT %MX25016.15 : BOOL;
	bArm1VertStn4Up_16 AT %MX25016.16 : BOOL;
	bArm1VertStn4Up_17 AT %MX25016.17 : BOOL;
	bArm1VertStn4Up_18 AT %MX25016.18 : BOOL;
	bArm1VertStn4Up_19 AT %MX25016.19 : BOOL;
	bArm1VertStn4Up_20 AT %MX25016.20 : BOOL;
	bArm1VertStn4Up_21 AT %MX25016.21 : BOOL;
	bArm1VertStn4Up_22 AT %MX25016.22 : BOOL;
	bArm1VertStn4Up_23 AT %MX25016.23 : BOOL;
	bArm1VertStn4Up_24 AT %MX25016.24 : BOOL;
	bArm1VertStn4Up_25 AT %MX25016.25 : BOOL;
	bArm1VertStn4Up_26 AT %MX25016.26 : BOOL;
	bArm1VertStn4Up_27 AT %MX25016.27 : BOOL;
	bArm1VertStn4Up_28 AT %MX25016.28 : BOOL;
	bArm1VertStn4Up_29 AT %MX25016.29 : BOOL;
	bArm1VertStn4Up_30 AT %MX25016.30 : BOOL;
	bArm1VertStn4Up_31 AT %MX25016.31 : BOOL;

	bArm1VertStn5Up_00 AT %MX25020.0 : BOOL;
	bArm1VertStn5Up_01 AT %MX25020.1 : BOOL;
	bArm1VertStn5Up_02 AT %MX25020.2 : BOOL;
	bArm1VertStn5Up_03 AT %MX25020.3 : BOOL;
	bArm1VertStn5Up_04 AT %MX25020.4 : BOOL;
	bArm1VertStn5Up_05 AT %MX25020.5 : BOOL;
	bArm1VertStn5Up_06 AT %MX25020.6 : BOOL;
	bArm1VertStn5Up_07 AT %MX25020.7 : BOOL;
	bArm1VertStn5Up_08 AT %MX25020.8 : BOOL;
	bArm1VertStn5Up_09 AT %MX25020.9 : BOOL;
	bArm1VertStn5Up_10 AT %MX25020.10 : BOOL;
	bArm1VertStn5Up_11 AT %MX25020.11 : BOOL;
	bArm1VertStn5Up_12 AT %MX25020.12 : BOOL;
	bArm1VertStn5Up_13 AT %MX25020.13 : BOOL;
	bArm1VertStn5Up_14 AT %MX25020.14 : BOOL;
	bArm1VertStn5Up_15 AT %MX25020.15 : BOOL;
	bArm1VertStn5Up_16 AT %MX25020.16 : BOOL;
	bArm1VertStn5Up_17 AT %MX25020.17 : BOOL;
	bArm1VertStn5Up_18 AT %MX25020.18 : BOOL;
	bArm1VertStn5Up_19 AT %MX25020.19 : BOOL;
	bArm1VertStn5Up_20 AT %MX25020.20 : BOOL;
	bArm1VertStn5Up_21 AT %MX25020.21 : BOOL;
	bArm1VertStn5Up_22 AT %MX25020.22 : BOOL;
	bArm1VertStn5Up_23 AT %MX25020.23 : BOOL;
	bArm1VertStn5Up_24 AT %MX25020.24 : BOOL;
	bArm1VertStn5Up_25 AT %MX25020.25 : BOOL;
	bArm1VertStn5Up_26 AT %MX25020.26 : BOOL;
	bArm1VertStn5Up_27 AT %MX25020.27 : BOOL;
	bArm1VertStn5Up_28 AT %MX25020.28 : BOOL;
	bArm1VertStn5Up_29 AT %MX25020.29 : BOOL;
	bArm1VertStn5Up_30 AT %MX25020.30 : BOOL;
	bArm1VertStn5Up_31 AT %MX25020.31 : BOOL;

	bArm1VertStn6Up_00 AT %MX25024.0 : BOOL;
	bArm1VertStn6Up_01 AT %MX25024.1 : BOOL;
	bArm1VertStn6Up_02 AT %MX25024.2 : BOOL;
	bArm1VertStn6Up_03 AT %MX25024.3 : BOOL;
	bArm1VertStn6Up_04 AT %MX25024.4 : BOOL;
	bArm1VertStn6Up_05 AT %MX25024.5 : BOOL;
	bArm1VertStn6Up_06 AT %MX25024.6 : BOOL;
	bArm1VertStn6Up_07 AT %MX25024.7 : BOOL;
	bArm1VertStn6Up_08 AT %MX25024.8 : BOOL;
	bArm1VertStn6Up_09 AT %MX25024.9 : BOOL;
	bArm1VertStn6Up_10 AT %MX25024.10 : BOOL;
	bArm1VertStn6Up_11 AT %MX25024.11 : BOOL;
	bArm1VertStn6Up_12 AT %MX25024.12 : BOOL;
	bArm1VertStn6Up_13 AT %MX25024.13 : BOOL;
	bArm1VertStn6Up_14 AT %MX25024.14 : BOOL;
	bArm1VertStn6Up_15 AT %MX25024.15 : BOOL;
	bArm1VertStn6Up_16 AT %MX25024.16 : BOOL;
	bArm1VertStn6Up_17 AT %MX25024.17 : BOOL;
	bArm1VertStn6Up_18 AT %MX25024.18 : BOOL;
	bArm1VertStn6Up_19 AT %MX25024.19 : BOOL;
	bArm1VertStn6Up_20 AT %MX25024.20 : BOOL;
	bArm1VertStn6Up_21 AT %MX25024.21 : BOOL;
	bArm1VertStn6Up_22 AT %MX25024.22 : BOOL;
	bArm1VertStn6Up_23 AT %MX25024.23 : BOOL;
	bArm1VertStn6Up_24 AT %MX25024.24 : BOOL;
	bArm1VertStn6Up_25 AT %MX25024.25 : BOOL;
	bArm1VertStn6Up_26 AT %MX25024.26 : BOOL;
	bArm1VertStn6Up_27 AT %MX25024.27 : BOOL;
	bArm1VertStn6Up_28 AT %MX25024.28 : BOOL;
	bArm1VertStn6Up_29 AT %MX25024.29 : BOOL;
	bArm1VertStn6Up_30 AT %MX25024.30 : BOOL;
	bArm1VertStn6Up_31 AT %MX25024.31 : BOOL;

	bArm1VertStn7Up_00 AT %MX25028.0 : BOOL;
	bArm1VertStn7Up_01 AT %MX25028.1 : BOOL;
	bArm1VertStn7Up_02 AT %MX25028.2 : BOOL;
	bArm1VertStn7Up_03 AT %MX25028.3 : BOOL;
	bArm1VertStn7Up_04 AT %MX25028.4 : BOOL;
	bArm1VertStn7Up_05 AT %MX25028.5 : BOOL;
	bArm1VertStn7Up_06 AT %MX25028.6 : BOOL;
	bArm1VertStn7Up_07 AT %MX25028.7 : BOOL;
	bArm1VertStn7Up_08 AT %MX25028.8 : BOOL;
	bArm1VertStn7Up_09 AT %MX25028.9 : BOOL;
	bArm1VertStn7Up_10 AT %MX25028.10 : BOOL;
	bArm1VertStn7Up_11 AT %MX25028.11 : BOOL;
	bArm1VertStn7Up_12 AT %MX25028.12 : BOOL;
	bArm1VertStn7Up_13 AT %MX25028.13 : BOOL;
	bArm1VertStn7Up_14 AT %MX25028.14 : BOOL;
	bArm1VertStn7Up_15 AT %MX25028.15 : BOOL;
	bArm1VertStn7Up_16 AT %MX25028.16 : BOOL;
	bArm1VertStn7Up_17 AT %MX25028.17 : BOOL;
	bArm1VertStn7Up_18 AT %MX25028.18 : BOOL;
	bArm1VertStn7Up_19 AT %MX25028.19 : BOOL;
	bArm1VertStn7Up_20 AT %MX25028.20 : BOOL;
	bArm1VertStn7Up_21 AT %MX25028.21 : BOOL;
	bArm1VertStn7Up_22 AT %MX25028.22 : BOOL;
	bArm1VertStn7Up_23 AT %MX25028.23 : BOOL;
	bArm1VertStn7Up_24 AT %MX25028.24 : BOOL;
	bArm1VertStn7Up_25 AT %MX25028.25 : BOOL;
	bArm1VertStn7Up_26 AT %MX25028.26 : BOOL;
	bArm1VertStn7Up_27 AT %MX25028.27 : BOOL;
	bArm1VertStn7Up_28 AT %MX25028.28 : BOOL;
	bArm1VertStn7Up_29 AT %MX25028.29 : BOOL;
	bArm1VertStn7Up_30 AT %MX25028.30 : BOOL;
	bArm1VertStn7Up_31 AT %MX25028.31 : BOOL;

	bArm1VertStn8Up_00 AT %MX25032.0 : BOOL;
	bArm1VertStn8Up_01 AT %MX25032.1 : BOOL;
	bArm1VertStn8Up_02 AT %MX25032.2 : BOOL;
	bArm1VertStn8Up_03 AT %MX25032.3 : BOOL;
	bArm1VertStn8Up_04 AT %MX25032.4 : BOOL;
	bArm1VertStn8Up_05 AT %MX25032.5 : BOOL;
	bArm1VertStn8Up_06 AT %MX25032.6 : BOOL;
	bArm1VertStn8Up_07 AT %MX25032.7 : BOOL;
	bArm1VertStn8Up_08 AT %MX25032.8 : BOOL;
	bArm1VertStn8Up_09 AT %MX25032.9 : BOOL;
	bArm1VertStn8Up_10 AT %MX25032.10 : BOOL;
	bArm1VertStn8Up_11 AT %MX25032.11 : BOOL;
	bArm1VertStn8Up_12 AT %MX25032.12 : BOOL;
	bArm1VertStn8Up_13 AT %MX25032.13 : BOOL;
	bArm1VertStn8Up_14 AT %MX25032.14 : BOOL;
	bArm1VertStn8Up_15 AT %MX25032.15 : BOOL;
	bArm1VertStn8Up_16 AT %MX25032.16 : BOOL;
	bArm1VertStn8Up_17 AT %MX25032.17 : BOOL;
	bArm1VertStn8Up_18 AT %MX25032.18 : BOOL;
	bArm1VertStn8Up_19 AT %MX25032.19 : BOOL;
	bArm1VertStn8Up_20 AT %MX25032.20 : BOOL;
	bArm1VertStn8Up_21 AT %MX25032.21 : BOOL;
	bArm1VertStn8Up_22 AT %MX25032.22 : BOOL;
	bArm1VertStn8Up_23 AT %MX25032.23 : BOOL;
	bArm1VertStn8Up_24 AT %MX25032.24 : BOOL;
	bArm1VertStn8Up_25 AT %MX25032.25 : BOOL;
	bArm1VertStn8Up_26 AT %MX25032.26 : BOOL;
	bArm1VertStn8Up_27 AT %MX25032.27 : BOOL;
	bArm1VertStn8Up_28 AT %MX25032.28 : BOOL;
	bArm1VertStn8Up_29 AT %MX25032.29 : BOOL;
	bArm1VertStn8Up_30 AT %MX25032.30 : BOOL;
	bArm1VertStn8Up_31 AT %MX25032.31 : BOOL;

	bArm1VertStn9Up_00 AT %MX25036.0 : BOOL;
	bArm1VertStn9Up_01 AT %MX25036.1 : BOOL;
	bArm1VertStn9Up_02 AT %MX25036.2 : BOOL;
	bArm1VertStn9Up_03 AT %MX25036.3 : BOOL;
	bArm1VertStn9Up_04 AT %MX25036.4 : BOOL;
	bArm1VertStn9Up_05 AT %MX25036.5 : BOOL;
	bArm1VertStn9Up_06 AT %MX25036.6 : BOOL;
	bArm1VertStn9Up_07 AT %MX25036.7 : BOOL;
	bArm1VertStn9Up_08 AT %MX25036.8 : BOOL;
	bArm1VertStn9Up_09 AT %MX25036.9 : BOOL;
	bArm1VertStn9Up_10 AT %MX25036.10 : BOOL;
	bArm1VertStn9Up_11 AT %MX25036.11 : BOOL;
	bArm1VertStn9Up_12 AT %MX25036.12 : BOOL;
	bArm1VertStn9Up_13 AT %MX25036.13 : BOOL;
	bArm1VertStn9Up_14 AT %MX25036.14 : BOOL;
	bArm1VertStn9Up_15 AT %MX25036.15 : BOOL;
	bArm1VertStn9Up_16 AT %MX25036.16 : BOOL;
	bArm1VertStn9Up_17 AT %MX25036.17 : BOOL;
	bArm1VertStn9Up_18 AT %MX25036.18 : BOOL;
	bArm1VertStn9Up_19 AT %MX25036.19 : BOOL;
	bArm1VertStn9Up_20 AT %MX25036.20 : BOOL;
	bArm1VertStn9Up_21 AT %MX25036.21 : BOOL;
	bArm1VertStn9Up_22 AT %MX25036.22 : BOOL;
	bArm1VertStn9Up_23 AT %MX25036.23 : BOOL;
	bArm1VertStn9Up_24 AT %MX25036.24 : BOOL;
	bArm1VertStn9Up_25 AT %MX25036.25 : BOOL;
	bArm1VertStn9Up_26 AT %MX25036.26 : BOOL;
	bArm1VertStn9Up_27 AT %MX25036.27 : BOOL;
	bArm1VertStn9Up_28 AT %MX25036.28 : BOOL;
	bArm1VertStn9Up_29 AT %MX25036.29 : BOOL;
	bArm1VertStn9Up_30 AT %MX25036.30 : BOOL;
	bArm1VertStn9Up_31 AT %MX25036.31 : BOOL;

	bArm1VertStn10Up_00 AT %MX25040.0 : BOOL;
	bArm1VertStn10Up_01 AT %MX25040.1 : BOOL;
	bArm1VertStn10Up_02 AT %MX25040.2 : BOOL;
	bArm1VertStn10Up_03 AT %MX25040.3 : BOOL;
	bArm1VertStn10Up_04 AT %MX25040.4 : BOOL;
	bArm1VertStn10Up_05 AT %MX25040.5 : BOOL;
	bArm1VertStn10Up_06 AT %MX25040.6 : BOOL;
	bArm1VertStn10Up_07 AT %MX25040.7 : BOOL;
	bArm1VertStn10Up_08 AT %MX25040.8 : BOOL;
	bArm1VertStn10Up_09 AT %MX25040.9 : BOOL;
	bArm1VertStn10Up_10 AT %MX25040.10 : BOOL;
	bArm1VertStn10Up_11 AT %MX25040.11 : BOOL;
	bArm1VertStn10Up_12 AT %MX25040.12 : BOOL;
	bArm1VertStn10Up_13 AT %MX25040.13 : BOOL;
	bArm1VertStn10Up_14 AT %MX25040.14 : BOOL;
	bArm1VertStn10Up_15 AT %MX25040.15 : BOOL;
	bArm1VertStn10Up_16 AT %MX25040.16 : BOOL;
	bArm1VertStn10Up_17 AT %MX25040.17 : BOOL;
	bArm1VertStn10Up_18 AT %MX25040.18 : BOOL;
	bArm1VertStn10Up_19 AT %MX25040.19 : BOOL;
	bArm1VertStn10Up_20 AT %MX25040.20 : BOOL;
	bArm1VertStn10Up_21 AT %MX25040.21 : BOOL;
	bArm1VertStn10Up_22 AT %MX25040.22 : BOOL;
	bArm1VertStn10Up_23 AT %MX25040.23 : BOOL;
	bArm1VertStn10Up_24 AT %MX25040.24 : BOOL;
	bArm1VertStn10Up_25 AT %MX25040.25 : BOOL;
	bArm1VertStn10Up_26 AT %MX25040.26 : BOOL;
	bArm1VertStn10Up_27 AT %MX25040.27 : BOOL;
	bArm1VertStn10Up_28 AT %MX25040.28 : BOOL;
	bArm1VertStn10Up_29 AT %MX25040.29 : BOOL;
	bArm1VertStn10Up_30 AT %MX25040.30 : BOOL;
	bArm1VertStn10Up_31 AT %MX25040.31 : BOOL;

	bArm1VertStn11Up_00 AT %MX25044.0 : BOOL;
	bArm1VertStn11Up_01 AT %MX25044.1 : BOOL;
	bArm1VertStn11Up_02 AT %MX25044.2 : BOOL;
	bArm1VertStn11Up_03 AT %MX25044.3 : BOOL;
	bArm1VertStn11Up_04 AT %MX25044.4 : BOOL;
	bArm1VertStn11Up_05 AT %MX25044.5 : BOOL;
	bArm1VertStn11Up_06 AT %MX25044.6 : BOOL;
	bArm1VertStn11Up_07 AT %MX25044.7 : BOOL;
	bArm1VertStn11Up_08 AT %MX25044.8 : BOOL;
	bArm1VertStn11Up_09 AT %MX25044.9 : BOOL;
	bArm1VertStn11Up_10 AT %MX25044.10 : BOOL;
	bArm1VertStn11Up_11 AT %MX25044.11 : BOOL;
	bArm1VertStn11Up_12 AT %MX25044.12 : BOOL;
	bArm1VertStn11Up_13 AT %MX25044.13 : BOOL;
	bArm1VertStn11Up_14 AT %MX25044.14 : BOOL;
	bArm1VertStn11Up_15 AT %MX25044.15 : BOOL;
	bArm1VertStn11Up_16 AT %MX25044.16 : BOOL;
	bArm1VertStn11Up_17 AT %MX25044.17 : BOOL;
	bArm1VertStn11Up_18 AT %MX25044.18 : BOOL;
	bArm1VertStn11Up_19 AT %MX25044.19 : BOOL;
	bArm1VertStn11Up_20 AT %MX25044.20 : BOOL;
	bArm1VertStn11Up_21 AT %MX25044.21 : BOOL;
	bArm1VertStn11Up_22 AT %MX25044.22 : BOOL;
	bArm1VertStn11Up_23 AT %MX25044.23 : BOOL;
	bArm1VertStn11Up_24 AT %MX25044.24 : BOOL;
	bArm1VertStn11Up_25 AT %MX25044.25 : BOOL;
	bArm1VertStn11Up_26 AT %MX25044.26 : BOOL;
	bArm1VertStn11Up_27 AT %MX25044.27 : BOOL;
	bArm1VertStn11Up_28 AT %MX25044.28 : BOOL;
	bArm1VertStn11Up_29 AT %MX25044.29 : BOOL;
	bArm1VertStn11Up_30 AT %MX25044.30 : BOOL;
	bArm1VertStn11Up_31 AT %MX25044.31 : BOOL;

	bArm1VertStn12Up_00 AT %MX25048.0 : BOOL;
	bArm1VertStn12Up_01 AT %MX25048.1 : BOOL;
	bArm1VertStn12Up_02 AT %MX25048.2 : BOOL;
	bArm1VertStn12Up_03 AT %MX25048.3 : BOOL;
	bArm1VertStn12Up_04 AT %MX25048.4 : BOOL;
	bArm1VertStn12Up_05 AT %MX25048.5 : BOOL;
	bArm1VertStn12Up_06 AT %MX25048.6 : BOOL;
	bArm1VertStn12Up_07 AT %MX25048.7 : BOOL;
	bArm1VertStn12Up_08 AT %MX25048.8 : BOOL;
	bArm1VertStn12Up_09 AT %MX25048.9 : BOOL;
	bArm1VertStn12Up_10 AT %MX25048.10 : BOOL;
	bArm1VertStn12Up_11 AT %MX25048.11 : BOOL;
	bArm1VertStn12Up_12 AT %MX25048.12 : BOOL;
	bArm1VertStn12Up_13 AT %MX25048.13 : BOOL;
	bArm1VertStn12Up_14 AT %MX25048.14 : BOOL;
	bArm1VertStn12Up_15 AT %MX25048.15 : BOOL;
	bArm1VertStn12Up_16 AT %MX25048.16 : BOOL;
	bArm1VertStn12Up_17 AT %MX25048.17 : BOOL;
	bArm1VertStn12Up_18 AT %MX25048.18 : BOOL;
	bArm1VertStn12Up_19 AT %MX25048.19 : BOOL;
	bArm1VertStn12Up_20 AT %MX25048.20 : BOOL;
	bArm1VertStn12Up_21 AT %MX25048.21 : BOOL;
	bArm1VertStn12Up_22 AT %MX25048.22 : BOOL;
	bArm1VertStn12Up_23 AT %MX25048.23 : BOOL;
	bArm1VertStn12Up_24 AT %MX25048.24 : BOOL;
	bArm1VertStn12Up_25 AT %MX25048.25 : BOOL;
	bArm1VertStn12Up_26 AT %MX25048.26 : BOOL;
	bArm1VertStn12Up_27 AT %MX25048.27 : BOOL;
	bArm1VertStn12Up_28 AT %MX25048.28 : BOOL;
	bArm1VertStn12Up_29 AT %MX25048.29 : BOOL;
	bArm1VertStn12Up_30 AT %MX25048.30 : BOOL;
	bArm1VertStn12Up_31 AT %MX25048.31 : BOOL;


(* xxxxxxxxxxxxxxxxxxxxxxxxxxxxxxxxxxxxxxx Vert xxxxxxxxxxxxxxxxxxxxxxxxxxxxxxxxxxxxxxx*)
(*========= Down SpSlanted BOOL LINK with %MX25100-MX25199 =========*)

	bArm1VertStn1SpSlanted_00 AT %MX25104.0 : BOOL;
	bArm1VertStn1SpSlanted_01 AT %MX25104.1 : BOOL;
	bArm1VertStn1SpSlanted_02 AT %MX25104.2 : BOOL;
	bArm1VertStn1SpSlanted_03 AT %MX25104.3 : BOOL;
	bArm1VertStn1SpSlanted_04 AT %MX25104.4 : BOOL;
	bArm1VertStn1SpSlanted_05 AT %MX25104.5 : BOOL;
	bArm1VertStn1SpSlanted_06 AT %MX25104.6 : BOOL;
	bArm1VertStn1SpSlanted_07 AT %MX25104.7 : BOOL;
	bArm1VertStn1SpSlanted_08 AT %MX25104.8 : BOOL;
	bArm1VertStn1SpSlanted_09 AT %MX25104.9 : BOOL;
	bArm1VertStn1SpSlanted_10 AT %MX25104.10 : BOOL;
	bArm1VertStn1SpSlanted_11 AT %MX25104.11 : BOOL;
	bArm1VertStn1SpSlanted_12 AT %MX25104.12 : BOOL;
	bArm1VertStn1SpSlanted_13 AT %MX25104.13 : BOOL;
	bArm1VertStn1SpSlanted_14 AT %MX25104.14 : BOOL;
	bArm1VertStn1SpSlanted_15 AT %MX25104.15 : BOOL;
	bArm1VertStn1SpSlanted_16 AT %MX25104.16 : BOOL;
	bArm1VertStn1SpSlanted_17 AT %MX25104.17 : BOOL;
	bArm1VertStn1SpSlanted_18 AT %MX25104.18 : BOOL;
	bArm1VertStn1SpSlanted_19 AT %MX25104.19 : BOOL;
	bArm1VertStn1SpSlanted_20 AT %MX25104.20 : BOOL;
	bArm1VertStn1SpSlanted_21 AT %MX25104.21 : BOOL;
	bArm1VertStn1SpSlanted_22 AT %MX25104.22 : BOOL;
	bArm1VertStn1SpSlanted_23 AT %MX25104.23 : BOOL;
	bArm1VertStn1SpSlanted_24 AT %MX25104.24 : BOOL;
	bArm1VertStn1SpSlanted_25 AT %MX25104.25 : BOOL;
	bArm1VertStn1SpSlanted_26 AT %MX25104.26 : BOOL;
	bArm1VertStn1SpSlanted_27 AT %MX25104.27 : BOOL;
	bArm1VertStn1SpSlanted_28 AT %MX25104.28 : BOOL;
	bArm1VertStn1SpSlanted_29 AT %MX25104.29 : BOOL;
	bArm1VertStn1SpSlanted_30 AT %MX25104.30 : BOOL;
	bArm1VertStn1SpSlanted_31 AT %MX25104.31 : BOOL;

	bArm1VertStn2SpSlanted_00 AT %MX25108.0 : BOOL;
	bArm1VertStn2SpSlanted_01 AT %MX25108.1 : BOOL;
	bArm1VertStn2SpSlanted_02 AT %MX25108.2 : BOOL;
	bArm1VertStn2SpSlanted_03 AT %MX25108.3 : BOOL;
	bArm1VertStn2SpSlanted_04 AT %MX25108.4 : BOOL;
	bArm1VertStn2SpSlanted_05 AT %MX25108.5 : BOOL;
	bArm1VertStn2SpSlanted_06 AT %MX25108.6 : BOOL;
	bArm1VertStn2SpSlanted_07 AT %MX25108.7 : BOOL;
	bArm1VertStn2SpSlanted_08 AT %MX25108.8 : BOOL;
	bArm1VertStn2SpSlanted_09 AT %MX25108.9 : BOOL;
	bArm1VertStn2SpSlanted_10 AT %MX25108.10 : BOOL;
	bArm1VertStn2SpSlanted_11 AT %MX25108.11 : BOOL;
	bArm1VertStn2SpSlanted_12 AT %MX25108.12 : BOOL;
	bArm1VertStn2SpSlanted_13 AT %MX25108.13 : BOOL;
	bArm1VertStn2SpSlanted_14 AT %MX25108.14 : BOOL;
	bArm1VertStn2SpSlanted_15 AT %MX25108.15 : BOOL;
	bArm1VertStn2SpSlanted_16 AT %MX25108.16 : BOOL;
	bArm1VertStn2SpSlanted_17 AT %MX25108.17 : BOOL;
	bArm1VertStn2SpSlanted_18 AT %MX25108.18 : BOOL;
	bArm1VertStn2SpSlanted_19 AT %MX25108.19 : BOOL;
	bArm1VertStn2SpSlanted_20 AT %MX25108.20 : BOOL;
	bArm1VertStn2SpSlanted_21 AT %MX25108.21 : BOOL;
	bArm1VertStn2SpSlanted_22 AT %MX25108.22 : BOOL;
	bArm1VertStn2SpSlanted_23 AT %MX25108.23 : BOOL;
	bArm1VertStn2SpSlanted_24 AT %MX25108.24 : BOOL;
	bArm1VertStn2SpSlanted_25 AT %MX25108.25 : BOOL;
	bArm1VertStn2SpSlanted_26 AT %MX25108.26 : BOOL;
	bArm1VertStn2SpSlanted_27 AT %MX25108.27 : BOOL;
	bArm1VertStn2SpSlanted_28 AT %MX25108.28 : BOOL;
	bArm1VertStn2SpSlanted_29 AT %MX25108.29 : BOOL;
	bArm1VertStn2SpSlanted_30 AT %MX25108.30 : BOOL;
	bArm1VertStn2SpSlanted_31 AT %MX25108.31 : BOOL;

	bArm1VertStn3SpSlanted_00 AT %MX25112.0 : BOOL;
	bArm1VertStn3SpSlanted_01 AT %MX25112.1 : BOOL;
	bArm1VertStn3SpSlanted_02 AT %MX25112.2 : BOOL;
	bArm1VertStn3SpSlanted_03 AT %MX25112.3 : BOOL;
	bArm1VertStn3SpSlanted_04 AT %MX25112.4 : BOOL;
	bArm1VertStn3SpSlanted_05 AT %MX25112.5 : BOOL;
	bArm1VertStn3SpSlanted_06 AT %MX25112.6 : BOOL;
	bArm1VertStn3SpSlanted_07 AT %MX25112.7 : BOOL;
	bArm1VertStn3SpSlanted_08 AT %MX25112.8 : BOOL;
	bArm1VertStn3SpSlanted_09 AT %MX25112.9 : BOOL;
	bArm1VertStn3SpSlanted_10 AT %MX25112.10 : BOOL;
	bArm1VertStn3SpSlanted_11 AT %MX25112.11 : BOOL;
	bArm1VertStn3SpSlanted_12 AT %MX25112.12 : BOOL;
	bArm1VertStn3SpSlanted_13 AT %MX25112.13 : BOOL;
	bArm1VertStn3SpSlanted_14 AT %MX25112.14 : BOOL;
	bArm1VertStn3SpSlanted_15 AT %MX25112.15 : BOOL;
	bArm1VertStn3SpSlanted_16 AT %MX25112.16 : BOOL;
	bArm1VertStn3SpSlanted_17 AT %MX25112.17 : BOOL;
	bArm1VertStn3SpSlanted_18 AT %MX25112.18 : BOOL;
	bArm1VertStn3SpSlanted_19 AT %MX25112.19 : BOOL;
	bArm1VertStn3SpSlanted_20 AT %MX25112.20 : BOOL;
	bArm1VertStn3SpSlanted_21 AT %MX25112.21 : BOOL;
	bArm1VertStn3SpSlanted_22 AT %MX25112.22 : BOOL;
	bArm1VertStn3SpSlanted_23 AT %MX25112.23 : BOOL;
	bArm1VertStn3SpSlanted_24 AT %MX25112.24 : BOOL;
	bArm1VertStn3SpSlanted_25 AT %MX25112.25 : BOOL;
	bArm1VertStn3SpSlanted_26 AT %MX25112.26 : BOOL;
	bArm1VertStn3SpSlanted_27 AT %MX25112.27 : BOOL;
	bArm1VertStn3SpSlanted_28 AT %MX25112.28 : BOOL;
	bArm1VertStn3SpSlanted_29 AT %MX25112.29 : BOOL;
	bArm1VertStn3SpSlanted_30 AT %MX25112.30 : BOOL;
	bArm1VertStn3SpSlanted_31 AT %MX25112.31 : BOOL;

	bArm1VertStn4SpSlanted_00 AT %MX25116.0 : BOOL;
	bArm1VertStn4SpSlanted_01 AT %MX25116.1 : BOOL;
	bArm1VertStn4SpSlanted_02 AT %MX25116.2 : BOOL;
	bArm1VertStn4SpSlanted_03 AT %MX25116.3 : BOOL;
	bArm1VertStn4SpSlanted_04 AT %MX25116.4 : BOOL;
	bArm1VertStn4SpSlanted_05 AT %MX25116.5 : BOOL;
	bArm1VertStn4SpSlanted_06 AT %MX25116.6 : BOOL;
	bArm1VertStn4SpSlanted_07 AT %MX25116.7 : BOOL;
	bArm1VertStn4SpSlanted_08 AT %MX25116.8 : BOOL;
	bArm1VertStn4SpSlanted_09 AT %MX25116.9 : BOOL;
	bArm1VertStn4SpSlanted_10 AT %MX25116.10 : BOOL;
	bArm1VertStn4SpSlanted_11 AT %MX25116.11 : BOOL;
	bArm1VertStn4SpSlanted_12 AT %MX25116.12 : BOOL;
	bArm1VertStn4SpSlanted_13 AT %MX25116.13 : BOOL;
	bArm1VertStn4SpSlanted_14 AT %MX25116.14 : BOOL;
	bArm1VertStn4SpSlanted_15 AT %MX25116.15 : BOOL;
	bArm1VertStn4SpSlanted_16 AT %MX25116.16 : BOOL;
	bArm1VertStn4SpSlanted_17 AT %MX25116.17 : BOOL;
	bArm1VertStn4SpSlanted_18 AT %MX25116.18 : BOOL;
	bArm1VertStn4SpSlanted_19 AT %MX25116.19 : BOOL;
	bArm1VertStn4SpSlanted_20 AT %MX25116.20 : BOOL;
	bArm1VertStn4SpSlanted_21 AT %MX25116.21 : BOOL;
	bArm1VertStn4SpSlanted_22 AT %MX25116.22 : BOOL;
	bArm1VertStn4SpSlanted_23 AT %MX25116.23 : BOOL;
	bArm1VertStn4SpSlanted_24 AT %MX25116.24 : BOOL;
	bArm1VertStn4SpSlanted_25 AT %MX25116.25 : BOOL;
	bArm1VertStn4SpSlanted_26 AT %MX25116.26 : BOOL;
	bArm1VertStn4SpSlanted_27 AT %MX25116.27 : BOOL;
	bArm1VertStn4SpSlanted_28 AT %MX25116.28 : BOOL;
	bArm1VertStn4SpSlanted_29 AT %MX25116.29 : BOOL;
	bArm1VertStn4SpSlanted_30 AT %MX25116.30 : BOOL;
	bArm1VertStn4SpSlanted_31 AT %MX25116.31 : BOOL;

	bArm1VertStn5SpSlanted_00 AT %MX25120.0 : BOOL;
	bArm1VertStn5SpSlanted_01 AT %MX25120.1 : BOOL;
	bArm1VertStn5SpSlanted_02 AT %MX25120.2 : BOOL;
	bArm1VertStn5SpSlanted_03 AT %MX25120.3 : BOOL;
	bArm1VertStn5SpSlanted_04 AT %MX25120.4 : BOOL;
	bArm1VertStn5SpSlanted_05 AT %MX25120.5 : BOOL;
	bArm1VertStn5SpSlanted_06 AT %MX25120.6 : BOOL;
	bArm1VertStn5SpSlanted_07 AT %MX25120.7 : BOOL;
	bArm1VertStn5SpSlanted_08 AT %MX25120.8 : BOOL;
	bArm1VertStn5SpSlanted_09 AT %MX25120.9 : BOOL;
	bArm1VertStn5SpSlanted_10 AT %MX25120.10 : BOOL;
	bArm1VertStn5SpSlanted_11 AT %MX25120.11 : BOOL;
	bArm1VertStn5SpSlanted_12 AT %MX25120.12 : BOOL;
	bArm1VertStn5SpSlanted_13 AT %MX25120.13 : BOOL;
	bArm1VertStn5SpSlanted_14 AT %MX25120.14 : BOOL;
	bArm1VertStn5SpSlanted_15 AT %MX25120.15 : BOOL;
	bArm1VertStn5SpSlanted_16 AT %MX25120.16 : BOOL;
	bArm1VertStn5SpSlanted_17 AT %MX25120.17 : BOOL;
	bArm1VertStn5SpSlanted_18 AT %MX25120.18 : BOOL;
	bArm1VertStn5SpSlanted_19 AT %MX25120.19 : BOOL;
	bArm1VertStn5SpSlanted_20 AT %MX25120.20 : BOOL;
	bArm1VertStn5SpSlanted_21 AT %MX25120.21 : BOOL;
	bArm1VertStn5SpSlanted_22 AT %MX25120.22 : BOOL;
	bArm1VertStn5SpSlanted_23 AT %MX25120.23 : BOOL;
	bArm1VertStn5SpSlanted_24 AT %MX25120.24 : BOOL;
	bArm1VertStn5SpSlanted_25 AT %MX25120.25 : BOOL;
	bArm1VertStn5SpSlanted_26 AT %MX25120.26 : BOOL;
	bArm1VertStn5SpSlanted_27 AT %MX25120.27 : BOOL;
	bArm1VertStn5SpSlanted_28 AT %MX25120.28 : BOOL;
	bArm1VertStn5SpSlanted_29 AT %MX25120.29 : BOOL;
	bArm1VertStn5SpSlanted_30 AT %MX25120.30 : BOOL;
	bArm1VertStn5SpSlanted_31 AT %MX25120.31 : BOOL;

	bArm1VertStn6SpSlanted_00 AT %MX25124.0 : BOOL;
	bArm1VertStn6SpSlanted_01 AT %MX25124.1 : BOOL;
	bArm1VertStn6SpSlanted_02 AT %MX25124.2 : BOOL;
	bArm1VertStn6SpSlanted_03 AT %MX25124.3 : BOOL;
	bArm1VertStn6SpSlanted_04 AT %MX25124.4 : BOOL;
	bArm1VertStn6SpSlanted_05 AT %MX25124.5 : BOOL;
	bArm1VertStn6SpSlanted_06 AT %MX25124.6 : BOOL;
	bArm1VertStn6SpSlanted_07 AT %MX25124.7 : BOOL;
	bArm1VertStn6SpSlanted_08 AT %MX25124.8 : BOOL;
	bArm1VertStn6SpSlanted_09 AT %MX25124.9 : BOOL;
	bArm1VertStn6SpSlanted_10 AT %MX25124.10 : BOOL;
	bArm1VertStn6SpSlanted_11 AT %MX25124.11 : BOOL;
	bArm1VertStn6SpSlanted_12 AT %MX25124.12 : BOOL;
	bArm1VertStn6SpSlanted_13 AT %MX25124.13 : BOOL;
	bArm1VertStn6SpSlanted_14 AT %MX25124.14 : BOOL;
	bArm1VertStn6SpSlanted_15 AT %MX25124.15 : BOOL;
	bArm1VertStn6SpSlanted_16 AT %MX25124.16 : BOOL;
	bArm1VertStn6SpSlanted_17 AT %MX25124.17 : BOOL;
	bArm1VertStn6SpSlanted_18 AT %MX25124.18 : BOOL;
	bArm1VertStn6SpSlanted_19 AT %MX25124.19 : BOOL;
	bArm1VertStn6SpSlanted_20 AT %MX25124.20 : BOOL;
	bArm1VertStn6SpSlanted_21 AT %MX25124.21 : BOOL;
	bArm1VertStn6SpSlanted_22 AT %MX25124.22 : BOOL;
	bArm1VertStn6SpSlanted_23 AT %MX25124.23 : BOOL;
	bArm1VertStn6SpSlanted_24 AT %MX25124.24 : BOOL;
	bArm1VertStn6SpSlanted_25 AT %MX25124.25 : BOOL;
	bArm1VertStn6SpSlanted_26 AT %MX25124.26 : BOOL;
	bArm1VertStn6SpSlanted_27 AT %MX25124.27 : BOOL;
	bArm1VertStn6SpSlanted_28 AT %MX25124.28 : BOOL;
	bArm1VertStn6SpSlanted_29 AT %MX25124.29 : BOOL;
	bArm1VertStn6SpSlanted_30 AT %MX25124.30 : BOOL;
	bArm1VertStn6SpSlanted_31 AT %MX25124.31 : BOOL;

	bArm1VertStn7SpSlanted_00 AT %MX25128.0 : BOOL;
	bArm1VertStn7SpSlanted_01 AT %MX25128.1 : BOOL;
	bArm1VertStn7SpSlanted_02 AT %MX25128.2 : BOOL;
	bArm1VertStn7SpSlanted_03 AT %MX25128.3 : BOOL;
	bArm1VertStn7SpSlanted_04 AT %MX25128.4 : BOOL;
	bArm1VertStn7SpSlanted_05 AT %MX25128.5 : BOOL;
	bArm1VertStn7SpSlanted_06 AT %MX25128.6 : BOOL;
	bArm1VertStn7SpSlanted_07 AT %MX25128.7 : BOOL;
	bArm1VertStn7SpSlanted_08 AT %MX25128.8 : BOOL;
	bArm1VertStn7SpSlanted_09 AT %MX25128.9 : BOOL;
	bArm1VertStn7SpSlanted_10 AT %MX25128.10 : BOOL;
	bArm1VertStn7SpSlanted_11 AT %MX25128.11 : BOOL;
	bArm1VertStn7SpSlanted_12 AT %MX25128.12 : BOOL;
	bArm1VertStn7SpSlanted_13 AT %MX25128.13 : BOOL;
	bArm1VertStn7SpSlanted_14 AT %MX25128.14 : BOOL;
	bArm1VertStn7SpSlanted_15 AT %MX25128.15 : BOOL;
	bArm1VertStn7SpSlanted_16 AT %MX25128.16 : BOOL;
	bArm1VertStn7SpSlanted_17 AT %MX25128.17 : BOOL;
	bArm1VertStn7SpSlanted_18 AT %MX25128.18 : BOOL;
	bArm1VertStn7SpSlanted_19 AT %MX25128.19 : BOOL;
	bArm1VertStn7SpSlanted_20 AT %MX25128.20 : BOOL;
	bArm1VertStn7SpSlanted_21 AT %MX25128.21 : BOOL;
	bArm1VertStn7SpSlanted_22 AT %MX25128.22 : BOOL;
	bArm1VertStn7SpSlanted_23 AT %MX25128.23 : BOOL;
	bArm1VertStn7SpSlanted_24 AT %MX25128.24 : BOOL;
	bArm1VertStn7SpSlanted_25 AT %MX25128.25 : BOOL;
	bArm1VertStn7SpSlanted_26 AT %MX25128.26 : BOOL;
	bArm1VertStn7SpSlanted_27 AT %MX25128.27 : BOOL;
	bArm1VertStn7SpSlanted_28 AT %MX25128.28 : BOOL;
	bArm1VertStn7SpSlanted_29 AT %MX25128.29 : BOOL;
	bArm1VertStn7SpSlanted_30 AT %MX25128.30 : BOOL;
	bArm1VertStn7SpSlanted_31 AT %MX25128.31 : BOOL;

	bArm1VertStn8SpSlanted_00 AT %MX25132.0 : BOOL;
	bArm1VertStn8SpSlanted_01 AT %MX25132.1 : BOOL;
	bArm1VertStn8SpSlanted_02 AT %MX25132.2 : BOOL;
	bArm1VertStn8SpSlanted_03 AT %MX25132.3 : BOOL;
	bArm1VertStn8SpSlanted_04 AT %MX25132.4 : BOOL;
	bArm1VertStn8SpSlanted_05 AT %MX25132.5 : BOOL;
	bArm1VertStn8SpSlanted_06 AT %MX25132.6 : BOOL;
	bArm1VertStn8SpSlanted_07 AT %MX25132.7 : BOOL;
	bArm1VertStn8SpSlanted_08 AT %MX25132.8 : BOOL;
	bArm1VertStn8SpSlanted_09 AT %MX25132.9 : BOOL;
	bArm1VertStn8SpSlanted_10 AT %MX25132.10 : BOOL;
	bArm1VertStn8SpSlanted_11 AT %MX25132.11 : BOOL;
	bArm1VertStn8SpSlanted_12 AT %MX25132.12 : BOOL;
	bArm1VertStn8SpSlanted_13 AT %MX25132.13 : BOOL;
	bArm1VertStn8SpSlanted_14 AT %MX25132.14 : BOOL;
	bArm1VertStn8SpSlanted_15 AT %MX25132.15 : BOOL;
	bArm1VertStn8SpSlanted_16 AT %MX25132.16 : BOOL;
	bArm1VertStn8SpSlanted_17 AT %MX25132.17 : BOOL;
	bArm1VertStn8SpSlanted_18 AT %MX25132.18 : BOOL;
	bArm1VertStn8SpSlanted_19 AT %MX25132.19 : BOOL;
	bArm1VertStn8SpSlanted_20 AT %MX25132.20 : BOOL;
	bArm1VertStn8SpSlanted_21 AT %MX25132.21 : BOOL;
	bArm1VertStn8SpSlanted_22 AT %MX25132.22 : BOOL;
	bArm1VertStn8SpSlanted_23 AT %MX25132.23 : BOOL;
	bArm1VertStn8SpSlanted_24 AT %MX25132.24 : BOOL;
	bArm1VertStn8SpSlanted_25 AT %MX25132.25 : BOOL;
	bArm1VertStn8SpSlanted_26 AT %MX25132.26 : BOOL;
	bArm1VertStn8SpSlanted_27 AT %MX25132.27 : BOOL;
	bArm1VertStn8SpSlanted_28 AT %MX25132.28 : BOOL;
	bArm1VertStn8SpSlanted_29 AT %MX25132.29 : BOOL;
	bArm1VertStn8SpSlanted_30 AT %MX25132.30 : BOOL;
	bArm1VertStn8SpSlanted_31 AT %MX25132.31 : BOOL;

	bArm1VertStn9SpSlanted_00 AT %MX25136.0 : BOOL;
	bArm1VertStn9SpSlanted_01 AT %MX25136.1 : BOOL;
	bArm1VertStn9SpSlanted_02 AT %MX25136.2 : BOOL;
	bArm1VertStn9SpSlanted_03 AT %MX25136.3 : BOOL;
	bArm1VertStn9SpSlanted_04 AT %MX25136.4 : BOOL;
	bArm1VertStn9SpSlanted_05 AT %MX25136.5 : BOOL;
	bArm1VertStn9SpSlanted_06 AT %MX25136.6 : BOOL;
	bArm1VertStn9SpSlanted_07 AT %MX25136.7 : BOOL;
	bArm1VertStn9SpSlanted_08 AT %MX25136.8 : BOOL;
	bArm1VertStn9SpSlanted_09 AT %MX25136.9 : BOOL;
	bArm1VertStn9SpSlanted_10 AT %MX25136.10 : BOOL;
	bArm1VertStn9SpSlanted_11 AT %MX25136.11 : BOOL;
	bArm1VertStn9SpSlanted_12 AT %MX25136.12 : BOOL;
	bArm1VertStn9SpSlanted_13 AT %MX25136.13 : BOOL;
	bArm1VertStn9SpSlanted_14 AT %MX25136.14 : BOOL;
	bArm1VertStn9SpSlanted_15 AT %MX25136.15 : BOOL;
	bArm1VertStn9SpSlanted_16 AT %MX25136.16 : BOOL;
	bArm1VertStn9SpSlanted_17 AT %MX25136.17 : BOOL;
	bArm1VertStn9SpSlanted_18 AT %MX25136.18 : BOOL;
	bArm1VertStn9SpSlanted_19 AT %MX25136.19 : BOOL;
	bArm1VertStn9SpSlanted_20 AT %MX25136.20 : BOOL;
	bArm1VertStn9SpSlanted_21 AT %MX25136.21 : BOOL;
	bArm1VertStn9SpSlanted_22 AT %MX25136.22 : BOOL;
	bArm1VertStn9SpSlanted_23 AT %MX25136.23 : BOOL;
	bArm1VertStn9SpSlanted_24 AT %MX25136.24 : BOOL;
	bArm1VertStn9SpSlanted_25 AT %MX25136.25 : BOOL;
	bArm1VertStn9SpSlanted_26 AT %MX25136.26 : BOOL;
	bArm1VertStn9SpSlanted_27 AT %MX25136.27 : BOOL;
	bArm1VertStn9SpSlanted_28 AT %MX25136.28 : BOOL;
	bArm1VertStn9SpSlanted_29 AT %MX25136.29 : BOOL;
	bArm1VertStn9SpSlanted_30 AT %MX25136.30 : BOOL;
	bArm1VertStn9SpSlanted_31 AT %MX25136.31 : BOOL;

	bArm1VertStn10SpSlanted_00 AT %MX25140.0 : BOOL;
	bArm1VertStn10SpSlanted_01 AT %MX25140.1 : BOOL;
	bArm1VertStn10SpSlanted_02 AT %MX25140.2 : BOOL;
	bArm1VertStn10SpSlanted_03 AT %MX25140.3 : BOOL;
	bArm1VertStn10SpSlanted_04 AT %MX25140.4 : BOOL;
	bArm1VertStn10SpSlanted_05 AT %MX25140.5 : BOOL;
	bArm1VertStn10SpSlanted_06 AT %MX25140.6 : BOOL;
	bArm1VertStn10SpSlanted_07 AT %MX25140.7 : BOOL;
	bArm1VertStn10SpSlanted_08 AT %MX25140.8 : BOOL;
	bArm1VertStn10SpSlanted_09 AT %MX25140.9 : BOOL;
	bArm1VertStn10SpSlanted_10 AT %MX25140.10 : BOOL;
	bArm1VertStn10SpSlanted_11 AT %MX25140.11 : BOOL;
	bArm1VertStn10SpSlanted_12 AT %MX25140.12 : BOOL;
	bArm1VertStn10SpSlanted_13 AT %MX25140.13 : BOOL;
	bArm1VertStn10SpSlanted_14 AT %MX25140.14 : BOOL;
	bArm1VertStn10SpSlanted_15 AT %MX25140.15 : BOOL;
	bArm1VertStn10SpSlanted_16 AT %MX25140.16 : BOOL;
	bArm1VertStn10SpSlanted_17 AT %MX25140.17 : BOOL;
	bArm1VertStn10SpSlanted_18 AT %MX25140.18 : BOOL;
	bArm1VertStn10SpSlanted_19 AT %MX25140.19 : BOOL;
	bArm1VertStn10SpSlanted_20 AT %MX25140.20 : BOOL;
	bArm1VertStn10SpSlanted_21 AT %MX25140.21 : BOOL;
	bArm1VertStn10SpSlanted_22 AT %MX25140.22 : BOOL;
	bArm1VertStn10SpSlanted_23 AT %MX25140.23 : BOOL;
	bArm1VertStn10SpSlanted_24 AT %MX25140.24 : BOOL;
	bArm1VertStn10SpSlanted_25 AT %MX25140.25 : BOOL;
	bArm1VertStn10SpSlanted_26 AT %MX25140.26 : BOOL;
	bArm1VertStn10SpSlanted_27 AT %MX25140.27 : BOOL;
	bArm1VertStn10SpSlanted_28 AT %MX25140.28 : BOOL;
	bArm1VertStn10SpSlanted_29 AT %MX25140.29 : BOOL;
	bArm1VertStn10SpSlanted_30 AT %MX25140.30 : BOOL;
	bArm1VertStn10SpSlanted_31 AT %MX25140.31 : BOOL;

	bArm1VertStn11SpSlanted_00 AT %MX25144.0 : BOOL;
	bArm1VertStn11SpSlanted_01 AT %MX25144.1 : BOOL;
	bArm1VertStn11SpSlanted_02 AT %MX25144.2 : BOOL;
	bArm1VertStn11SpSlanted_03 AT %MX25144.3 : BOOL;
	bArm1VertStn11SpSlanted_04 AT %MX25144.4 : BOOL;
	bArm1VertStn11SpSlanted_05 AT %MX25144.5 : BOOL;
	bArm1VertStn11SpSlanted_06 AT %MX25144.6 : BOOL;
	bArm1VertStn11SpSlanted_07 AT %MX25144.7 : BOOL;
	bArm1VertStn11SpSlanted_08 AT %MX25144.8 : BOOL;
	bArm1VertStn11SpSlanted_09 AT %MX25144.9 : BOOL;
	bArm1VertStn11SpSlanted_10 AT %MX25144.10 : BOOL;
	bArm1VertStn11SpSlanted_11 AT %MX25144.11 : BOOL;
	bArm1VertStn11SpSlanted_12 AT %MX25144.12 : BOOL;
	bArm1VertStn11SpSlanted_13 AT %MX25144.13 : BOOL;
	bArm1VertStn11SpSlanted_14 AT %MX25144.14 : BOOL;
	bArm1VertStn11SpSlanted_15 AT %MX25144.15 : BOOL;
	bArm1VertStn11SpSlanted_16 AT %MX25144.16 : BOOL;
	bArm1VertStn11SpSlanted_17 AT %MX25144.17 : BOOL;
	bArm1VertStn11SpSlanted_18 AT %MX25144.18 : BOOL;
	bArm1VertStn11SpSlanted_19 AT %MX25144.19 : BOOL;
	bArm1VertStn11SpSlanted_20 AT %MX25144.20 : BOOL;
	bArm1VertStn11SpSlanted_21 AT %MX25144.21 : BOOL;
	bArm1VertStn11SpSlanted_22 AT %MX25144.22 : BOOL;
	bArm1VertStn11SpSlanted_23 AT %MX25144.23 : BOOL;
	bArm1VertStn11SpSlanted_24 AT %MX25144.24 : BOOL;
	bArm1VertStn11SpSlanted_25 AT %MX25144.25 : BOOL;
	bArm1VertStn11SpSlanted_26 AT %MX25144.26 : BOOL;
	bArm1VertStn11SpSlanted_27 AT %MX25144.27 : BOOL;
	bArm1VertStn11SpSlanted_28 AT %MX25144.28 : BOOL;
	bArm1VertStn11SpSlanted_29 AT %MX25144.29 : BOOL;
	bArm1VertStn11SpSlanted_30 AT %MX25144.30 : BOOL;
	bArm1VertStn11SpSlanted_31 AT %MX25144.31 : BOOL;

	bArm1VertStn12SpSlanted_00 AT %MX25148.0 : BOOL;
	bArm1VertStn12SpSlanted_01 AT %MX25148.1 : BOOL;
	bArm1VertStn12SpSlanted_02 AT %MX25148.2 : BOOL;
	bArm1VertStn12SpSlanted_03 AT %MX25148.3 : BOOL;
	bArm1VertStn12SpSlanted_04 AT %MX25148.4 : BOOL;
	bArm1VertStn12SpSlanted_05 AT %MX25148.5 : BOOL;
	bArm1VertStn12SpSlanted_06 AT %MX25148.6 : BOOL;
	bArm1VertStn12SpSlanted_07 AT %MX25148.7 : BOOL;
	bArm1VertStn12SpSlanted_08 AT %MX25148.8 : BOOL;
	bArm1VertStn12SpSlanted_09 AT %MX25148.9 : BOOL;
	bArm1VertStn12SpSlanted_10 AT %MX25148.10 : BOOL;
	bArm1VertStn12SpSlanted_11 AT %MX25148.11 : BOOL;
	bArm1VertStn12SpSlanted_12 AT %MX25148.12 : BOOL;
	bArm1VertStn12SpSlanted_13 AT %MX25148.13 : BOOL;
	bArm1VertStn12SpSlanted_14 AT %MX25148.14 : BOOL;
	bArm1VertStn12SpSlanted_15 AT %MX25148.15 : BOOL;
	bArm1VertStn12SpSlanted_16 AT %MX25148.16 : BOOL;
	bArm1VertStn12SpSlanted_17 AT %MX25148.17 : BOOL;
	bArm1VertStn12SpSlanted_18 AT %MX25148.18 : BOOL;
	bArm1VertStn12SpSlanted_19 AT %MX25148.19 : BOOL;
	bArm1VertStn12SpSlanted_20 AT %MX25148.20 : BOOL;
	bArm1VertStn12SpSlanted_21 AT %MX25148.21 : BOOL;
	bArm1VertStn12SpSlanted_22 AT %MX25148.22 : BOOL;
	bArm1VertStn12SpSlanted_23 AT %MX25148.23 : BOOL;
	bArm1VertStn12SpSlanted_24 AT %MX25148.24 : BOOL;
	bArm1VertStn12SpSlanted_25 AT %MX25148.25 : BOOL;
	bArm1VertStn12SpSlanted_26 AT %MX25148.26 : BOOL;
	bArm1VertStn12SpSlanted_27 AT %MX25148.27 : BOOL;
	bArm1VertStn12SpSlanted_28 AT %MX25148.28 : BOOL;
	bArm1VertStn12SpSlanted_29 AT %MX25148.29 : BOOL;
	bArm1VertStn12SpSlanted_30 AT %MX25148.30 : BOOL;
	bArm1VertStn12SpSlanted_31 AT %MX25148.31 : BOOL;


(* xxxxxxxxxxxxxxxxxxxxxxxxxxxxxxxxxxxxxxx Vert xxxxxxxxxxxxxxxxxxxxxxxxxxxxxxxxxxxxxxx*)
(*========= Down Regular BOOL LINK with %MX25200-MX25299 =========*)

	bArm1VertStn1Regular_00 AT %MX25204.0 : BOOL;
	bArm1VertStn1Regular_01 AT %MX25204.1 : BOOL;
	bArm1VertStn1Regular_02 AT %MX25204.2 : BOOL;
	bArm1VertStn1Regular_03 AT %MX25204.3 : BOOL;
	bArm1VertStn1Regular_04 AT %MX25204.4 : BOOL;
	bArm1VertStn1Regular_05 AT %MX25204.5 : BOOL;
	bArm1VertStn1Regular_06 AT %MX25204.6 : BOOL;
	bArm1VertStn1Regular_07 AT %MX25204.7 : BOOL;
	bArm1VertStn1Regular_08 AT %MX25204.8 : BOOL;
	bArm1VertStn1Regular_09 AT %MX25204.9 : BOOL;
	bArm1VertStn1Regular_10 AT %MX25204.10 : BOOL;
	bArm1VertStn1Regular_11 AT %MX25204.11 : BOOL;
	bArm1VertStn1Regular_12 AT %MX25204.12 : BOOL;
	bArm1VertStn1Regular_13 AT %MX25204.13 : BOOL;
	bArm1VertStn1Regular_14 AT %MX25204.14 : BOOL;
	bArm1VertStn1Regular_15 AT %MX25204.15 : BOOL;
	bArm1VertStn1Regular_16 AT %MX25204.16 : BOOL;
	bArm1VertStn1Regular_17 AT %MX25204.17 : BOOL;
	bArm1VertStn1Regular_18 AT %MX25204.18 : BOOL;
	bArm1VertStn1Regular_19 AT %MX25204.19 : BOOL;
	bArm1VertStn1Regular_20 AT %MX25204.20 : BOOL;
	bArm1VertStn1Regular_21 AT %MX25204.21 : BOOL;
	bArm1VertStn1Regular_22 AT %MX25204.22 : BOOL;
	bArm1VertStn1Regular_23 AT %MX25204.23 : BOOL;
	bArm1VertStn1Regular_24 AT %MX25204.24 : BOOL;
	bArm1VertStn1Regular_25 AT %MX25204.25 : BOOL;
	bArm1VertStn1Regular_26 AT %MX25204.26 : BOOL;
	bArm1VertStn1Regular_27 AT %MX25204.27 : BOOL;
	bArm1VertStn1Regular_28 AT %MX25204.28 : BOOL;
	bArm1VertStn1Regular_29 AT %MX25204.29 : BOOL;
	bArm1VertStn1Regular_30 AT %MX25204.30 : BOOL;
	bArm1VertStn1Regular_31 AT %MX25204.31 : BOOL;

	bArm1VertStn2Regular_00 AT %MX25208.0 : BOOL;
	bArm1VertStn2Regular_01 AT %MX25208.1 : BOOL;
	bArm1VertStn2Regular_02 AT %MX25208.2 : BOOL;
	bArm1VertStn2Regular_03 AT %MX25208.3 : BOOL;
	bArm1VertStn2Regular_04 AT %MX25208.4 : BOOL;
	bArm1VertStn2Regular_05 AT %MX25208.5 : BOOL;
	bArm1VertStn2Regular_06 AT %MX25208.6 : BOOL;
	bArm1VertStn2Regular_07 AT %MX25208.7 : BOOL;
	bArm1VertStn2Regular_08 AT %MX25208.8 : BOOL;
	bArm1VertStn2Regular_09 AT %MX25208.9 : BOOL;
	bArm1VertStn2Regular_10 AT %MX25208.10 : BOOL;
	bArm1VertStn2Regular_11 AT %MX25208.11 : BOOL;
	bArm1VertStn2Regular_12 AT %MX25208.12 : BOOL;
	bArm1VertStn2Regular_13 AT %MX25208.13 : BOOL;
	bArm1VertStn2Regular_14 AT %MX25208.14 : BOOL;
	bArm1VertStn2Regular_15 AT %MX25208.15 : BOOL;
	bArm1VertStn2Regular_16 AT %MX25208.16 : BOOL;
	bArm1VertStn2Regular_17 AT %MX25208.17 : BOOL;
	bArm1VertStn2Regular_18 AT %MX25208.18 : BOOL;
	bArm1VertStn2Regular_19 AT %MX25208.19 : BOOL;
	bArm1VertStn2Regular_20 AT %MX25208.20 : BOOL;
	bArm1VertStn2Regular_21 AT %MX25208.21 : BOOL;
	bArm1VertStn2Regular_22 AT %MX25208.22 : BOOL;
	bArm1VertStn2Regular_23 AT %MX25208.23 : BOOL;
	bArm1VertStn2Regular_24 AT %MX25208.24 : BOOL;
	bArm1VertStn2Regular_25 AT %MX25208.25 : BOOL;
	bArm1VertStn2Regular_26 AT %MX25208.26 : BOOL;
	bArm1VertStn2Regular_27 AT %MX25208.27 : BOOL;
	bArm1VertStn2Regular_28 AT %MX25208.28 : BOOL;
	bArm1VertStn2Regular_29 AT %MX25208.29 : BOOL;
	bArm1VertStn2Regular_30 AT %MX25208.30 : BOOL;
	bArm1VertStn2Regular_31 AT %MX25208.31 : BOOL;

	bArm1VertStn3Regular_00 AT %MX25212.0 : BOOL;
	bArm1VertStn3Regular_01 AT %MX25212.1 : BOOL;
	bArm1VertStn3Regular_02 AT %MX25212.2 : BOOL;
	bArm1VertStn3Regular_03 AT %MX25212.3 : BOOL;
	bArm1VertStn3Regular_04 AT %MX25212.4 : BOOL;
	bArm1VertStn3Regular_05 AT %MX25212.5 : BOOL;
	bArm1VertStn3Regular_06 AT %MX25212.6 : BOOL;
	bArm1VertStn3Regular_07 AT %MX25212.7 : BOOL;
	bArm1VertStn3Regular_08 AT %MX25212.8 : BOOL;
	bArm1VertStn3Regular_09 AT %MX25212.9 : BOOL;
	bArm1VertStn3Regular_10 AT %MX25212.10 : BOOL;
	bArm1VertStn3Regular_11 AT %MX25212.11 : BOOL;
	bArm1VertStn3Regular_12 AT %MX25212.12 : BOOL;
	bArm1VertStn3Regular_13 AT %MX25212.13 : BOOL;
	bArm1VertStn3Regular_14 AT %MX25212.14 : BOOL;
	bArm1VertStn3Regular_15 AT %MX25212.15 : BOOL;
	bArm1VertStn3Regular_16 AT %MX25212.16 : BOOL;
	bArm1VertStn3Regular_17 AT %MX25212.17 : BOOL;
	bArm1VertStn3Regular_18 AT %MX25212.18 : BOOL;
	bArm1VertStn3Regular_19 AT %MX25212.19 : BOOL;
	bArm1VertStn3Regular_20 AT %MX25212.20 : BOOL;
	bArm1VertStn3Regular_21 AT %MX25212.21 : BOOL;
	bArm1VertStn3Regular_22 AT %MX25212.22 : BOOL;
	bArm1VertStn3Regular_23 AT %MX25212.23 : BOOL;
	bArm1VertStn3Regular_24 AT %MX25212.24 : BOOL;
	bArm1VertStn3Regular_25 AT %MX25212.25 : BOOL;
	bArm1VertStn3Regular_26 AT %MX25212.26 : BOOL;
	bArm1VertStn3Regular_27 AT %MX25212.27 : BOOL;
	bArm1VertStn3Regular_28 AT %MX25212.28 : BOOL;
	bArm1VertStn3Regular_29 AT %MX25212.29 : BOOL;
	bArm1VertStn3Regular_30 AT %MX25212.30 : BOOL;
	bArm1VertStn3Regular_31 AT %MX25212.31 : BOOL;

	bArm1VertStn4Regular_00 AT %MX25216.0 : BOOL;
	bArm1VertStn4Regular_01 AT %MX25216.1 : BOOL;
	bArm1VertStn4Regular_02 AT %MX25216.2 : BOOL;
	bArm1VertStn4Regular_03 AT %MX25216.3 : BOOL;
	bArm1VertStn4Regular_04 AT %MX25216.4 : BOOL;
	bArm1VertStn4Regular_05 AT %MX25216.5 : BOOL;
	bArm1VertStn4Regular_06 AT %MX25216.6 : BOOL;
	bArm1VertStn4Regular_07 AT %MX25216.7 : BOOL;
	bArm1VertStn4Regular_08 AT %MX25216.8 : BOOL;
	bArm1VertStn4Regular_09 AT %MX25216.9 : BOOL;
	bArm1VertStn4Regular_10 AT %MX25216.10 : BOOL;
	bArm1VertStn4Regular_11 AT %MX25216.11 : BOOL;
	bArm1VertStn4Regular_12 AT %MX25216.12 : BOOL;
	bArm1VertStn4Regular_13 AT %MX25216.13 : BOOL;
	bArm1VertStn4Regular_14 AT %MX25216.14 : BOOL;
	bArm1VertStn4Regular_15 AT %MX25216.15 : BOOL;
	bArm1VertStn4Regular_16 AT %MX25216.16 : BOOL;
	bArm1VertStn4Regular_17 AT %MX25216.17 : BOOL;
	bArm1VertStn4Regular_18 AT %MX25216.18 : BOOL;
	bArm1VertStn4Regular_19 AT %MX25216.19 : BOOL;
	bArm1VertStn4Regular_20 AT %MX25216.20 : BOOL;
	bArm1VertStn4Regular_21 AT %MX25216.21 : BOOL;
	bArm1VertStn4Regular_22 AT %MX25216.22 : BOOL;
	bArm1VertStn4Regular_23 AT %MX25216.23 : BOOL;
	bArm1VertStn4Regular_24 AT %MX25216.24 : BOOL;
	bArm1VertStn4Regular_25 AT %MX25216.25 : BOOL;
	bArm1VertStn4Regular_26 AT %MX25216.26 : BOOL;
	bArm1VertStn4Regular_27 AT %MX25216.27 : BOOL;
	bArm1VertStn4Regular_28 AT %MX25216.28 : BOOL;
	bArm1VertStn4Regular_29 AT %MX25216.29 : BOOL;
	bArm1VertStn4Regular_30 AT %MX25216.30 : BOOL;
	bArm1VertStn4Regular_31 AT %MX25216.31 : BOOL;

	bArm1VertStn5Regular_00 AT %MX25220.0 : BOOL;
	bArm1VertStn5Regular_01 AT %MX25220.1 : BOOL;
	bArm1VertStn5Regular_02 AT %MX25220.2 : BOOL;
	bArm1VertStn5Regular_03 AT %MX25220.3 : BOOL;
	bArm1VertStn5Regular_04 AT %MX25220.4 : BOOL;
	bArm1VertStn5Regular_05 AT %MX25220.5 : BOOL;
	bArm1VertStn5Regular_06 AT %MX25220.6 : BOOL;
	bArm1VertStn5Regular_07 AT %MX25220.7 : BOOL;
	bArm1VertStn5Regular_08 AT %MX25220.8 : BOOL;
	bArm1VertStn5Regular_09 AT %MX25220.9 : BOOL;
	bArm1VertStn5Regular_10 AT %MX25220.10 : BOOL;
	bArm1VertStn5Regular_11 AT %MX25220.11 : BOOL;
	bArm1VertStn5Regular_12 AT %MX25220.12 : BOOL;
	bArm1VertStn5Regular_13 AT %MX25220.13 : BOOL;
	bArm1VertStn5Regular_14 AT %MX25220.14 : BOOL;
	bArm1VertStn5Regular_15 AT %MX25220.15 : BOOL;
	bArm1VertStn5Regular_16 AT %MX25220.16 : BOOL;
	bArm1VertStn5Regular_17 AT %MX25220.17 : BOOL;
	bArm1VertStn5Regular_18 AT %MX25220.18 : BOOL;
	bArm1VertStn5Regular_19 AT %MX25220.19 : BOOL;
	bArm1VertStn5Regular_20 AT %MX25220.20 : BOOL;
	bArm1VertStn5Regular_21 AT %MX25220.21 : BOOL;
	bArm1VertStn5Regular_22 AT %MX25220.22 : BOOL;
	bArm1VertStn5Regular_23 AT %MX25220.23 : BOOL;
	bArm1VertStn5Regular_24 AT %MX25220.24 : BOOL;
	bArm1VertStn5Regular_25 AT %MX25220.25 : BOOL;
	bArm1VertStn5Regular_26 AT %MX25220.26 : BOOL;
	bArm1VertStn5Regular_27 AT %MX25220.27 : BOOL;
	bArm1VertStn5Regular_28 AT %MX25220.28 : BOOL;
	bArm1VertStn5Regular_29 AT %MX25220.29 : BOOL;
	bArm1VertStn5Regular_30 AT %MX25220.30 : BOOL;
	bArm1VertStn5Regular_31 AT %MX25220.31 : BOOL;

	bArm1VertStn6Regular_00 AT %MX25224.0 : BOOL;
	bArm1VertStn6Regular_01 AT %MX25224.1 : BOOL;
	bArm1VertStn6Regular_02 AT %MX25224.2 : BOOL;
	bArm1VertStn6Regular_03 AT %MX25224.3 : BOOL;
	bArm1VertStn6Regular_04 AT %MX25224.4 : BOOL;
	bArm1VertStn6Regular_05 AT %MX25224.5 : BOOL;
	bArm1VertStn6Regular_06 AT %MX25224.6 : BOOL;
	bArm1VertStn6Regular_07 AT %MX25224.7 : BOOL;
	bArm1VertStn6Regular_08 AT %MX25224.8 : BOOL;
	bArm1VertStn6Regular_09 AT %MX25224.9 : BOOL;
	bArm1VertStn6Regular_10 AT %MX25224.10 : BOOL;
	bArm1VertStn6Regular_11 AT %MX25224.11 : BOOL;
	bArm1VertStn6Regular_12 AT %MX25224.12 : BOOL;
	bArm1VertStn6Regular_13 AT %MX25224.13 : BOOL;
	bArm1VertStn6Regular_14 AT %MX25224.14 : BOOL;
	bArm1VertStn6Regular_15 AT %MX25224.15 : BOOL;
	bArm1VertStn6Regular_16 AT %MX25224.16 : BOOL;
	bArm1VertStn6Regular_17 AT %MX25224.17 : BOOL;
	bArm1VertStn6Regular_18 AT %MX25224.18 : BOOL;
	bArm1VertStn6Regular_19 AT %MX25224.19 : BOOL;
	bArm1VertStn6Regular_20 AT %MX25224.20 : BOOL;
	bArm1VertStn6Regular_21 AT %MX25224.21 : BOOL;
	bArm1VertStn6Regular_22 AT %MX25224.22 : BOOL;
	bArm1VertStn6Regular_23 AT %MX25224.23 : BOOL;
	bArm1VertStn6Regular_24 AT %MX25224.24 : BOOL;
	bArm1VertStn6Regular_25 AT %MX25224.25 : BOOL;
	bArm1VertStn6Regular_26 AT %MX25224.26 : BOOL;
	bArm1VertStn6Regular_27 AT %MX25224.27 : BOOL;
	bArm1VertStn6Regular_28 AT %MX25224.28 : BOOL;
	bArm1VertStn6Regular_29 AT %MX25224.29 : BOOL;
	bArm1VertStn6Regular_30 AT %MX25224.30 : BOOL;
	bArm1VertStn6Regular_31 AT %MX25224.31 : BOOL;

	bArm1VertStn7Regular_00 AT %MX25228.0 : BOOL;
	bArm1VertStn7Regular_01 AT %MX25228.1 : BOOL;
	bArm1VertStn7Regular_02 AT %MX25228.2 : BOOL;
	bArm1VertStn7Regular_03 AT %MX25228.3 : BOOL;
	bArm1VertStn7Regular_04 AT %MX25228.4 : BOOL;
	bArm1VertStn7Regular_05 AT %MX25228.5 : BOOL;
	bArm1VertStn7Regular_06 AT %MX25228.6 : BOOL;
	bArm1VertStn7Regular_07 AT %MX25228.7 : BOOL;
	bArm1VertStn7Regular_08 AT %MX25228.8 : BOOL;
	bArm1VertStn7Regular_09 AT %MX25228.9 : BOOL;
	bArm1VertStn7Regular_10 AT %MX25228.10 : BOOL;
	bArm1VertStn7Regular_11 AT %MX25228.11 : BOOL;
	bArm1VertStn7Regular_12 AT %MX25228.12 : BOOL;
	bArm1VertStn7Regular_13 AT %MX25228.13 : BOOL;
	bArm1VertStn7Regular_14 AT %MX25228.14 : BOOL;
	bArm1VertStn7Regular_15 AT %MX25228.15 : BOOL;
	bArm1VertStn7Regular_16 AT %MX25228.16 : BOOL;
	bArm1VertStn7Regular_17 AT %MX25228.17 : BOOL;
	bArm1VertStn7Regular_18 AT %MX25228.18 : BOOL;
	bArm1VertStn7Regular_19 AT %MX25228.19 : BOOL;
	bArm1VertStn7Regular_20 AT %MX25228.20 : BOOL;
	bArm1VertStn7Regular_21 AT %MX25228.21 : BOOL;
	bArm1VertStn7Regular_22 AT %MX25228.22 : BOOL;
	bArm1VertStn7Regular_23 AT %MX25228.23 : BOOL;
	bArm1VertStn7Regular_24 AT %MX25228.24 : BOOL;
	bArm1VertStn7Regular_25 AT %MX25228.25 : BOOL;
	bArm1VertStn7Regular_26 AT %MX25228.26 : BOOL;
	bArm1VertStn7Regular_27 AT %MX25228.27 : BOOL;
	bArm1VertStn7Regular_28 AT %MX25228.28 : BOOL;
	bArm1VertStn7Regular_29 AT %MX25228.29 : BOOL;
	bArm1VertStn7Regular_30 AT %MX25228.30 : BOOL;
	bArm1VertStn7Regular_31 AT %MX25228.31 : BOOL;

	bArm1VertStn8Regular_00 AT %MX25232.0 : BOOL;
	bArm1VertStn8Regular_01 AT %MX25232.1 : BOOL;
	bArm1VertStn8Regular_02 AT %MX25232.2 : BOOL;
	bArm1VertStn8Regular_03 AT %MX25232.3 : BOOL;
	bArm1VertStn8Regular_04 AT %MX25232.4 : BOOL;
	bArm1VertStn8Regular_05 AT %MX25232.5 : BOOL;
	bArm1VertStn8Regular_06 AT %MX25232.6 : BOOL;
	bArm1VertStn8Regular_07 AT %MX25232.7 : BOOL;
	bArm1VertStn8Regular_08 AT %MX25232.8 : BOOL;
	bArm1VertStn8Regular_09 AT %MX25232.9 : BOOL;
	bArm1VertStn8Regular_10 AT %MX25232.10 : BOOL;
	bArm1VertStn8Regular_11 AT %MX25232.11 : BOOL;
	bArm1VertStn8Regular_12 AT %MX25232.12 : BOOL;
	bArm1VertStn8Regular_13 AT %MX25232.13 : BOOL;
	bArm1VertStn8Regular_14 AT %MX25232.14 : BOOL;
	bArm1VertStn8Regular_15 AT %MX25232.15 : BOOL;
	bArm1VertStn8Regular_16 AT %MX25232.16 : BOOL;
	bArm1VertStn8Regular_17 AT %MX25232.17 : BOOL;
	bArm1VertStn8Regular_18 AT %MX25232.18 : BOOL;
	bArm1VertStn8Regular_19 AT %MX25232.19 : BOOL;
	bArm1VertStn8Regular_20 AT %MX25232.20 : BOOL;
	bArm1VertStn8Regular_21 AT %MX25232.21 : BOOL;
	bArm1VertStn8Regular_22 AT %MX25232.22 : BOOL;
	bArm1VertStn8Regular_23 AT %MX25232.23 : BOOL;
	bArm1VertStn8Regular_24 AT %MX25232.24 : BOOL;
	bArm1VertStn8Regular_25 AT %MX25232.25 : BOOL;
	bArm1VertStn8Regular_26 AT %MX25232.26 : BOOL;
	bArm1VertStn8Regular_27 AT %MX25232.27 : BOOL;
	bArm1VertStn8Regular_28 AT %MX25232.28 : BOOL;
	bArm1VertStn8Regular_29 AT %MX25232.29 : BOOL;
	bArm1VertStn8Regular_30 AT %MX25232.30 : BOOL;
	bArm1VertStn8Regular_31 AT %MX25232.31 : BOOL;

	bArm1VertStn9Regular_00 AT %MX25236.0 : BOOL;
	bArm1VertStn9Regular_01 AT %MX25236.1 : BOOL;
	bArm1VertStn9Regular_02 AT %MX25236.2 : BOOL;
	bArm1VertStn9Regular_03 AT %MX25236.3 : BOOL;
	bArm1VertStn9Regular_04 AT %MX25236.4 : BOOL;
	bArm1VertStn9Regular_05 AT %MX25236.5 : BOOL;
	bArm1VertStn9Regular_06 AT %MX25236.6 : BOOL;
	bArm1VertStn9Regular_07 AT %MX25236.7 : BOOL;
	bArm1VertStn9Regular_08 AT %MX25236.8 : BOOL;
	bArm1VertStn9Regular_09 AT %MX25236.9 : BOOL;
	bArm1VertStn9Regular_10 AT %MX25236.10 : BOOL;
	bArm1VertStn9Regular_11 AT %MX25236.11 : BOOL;
	bArm1VertStn9Regular_12 AT %MX25236.12 : BOOL;
	bArm1VertStn9Regular_13 AT %MX25236.13 : BOOL;
	bArm1VertStn9Regular_14 AT %MX25236.14 : BOOL;
	bArm1VertStn9Regular_15 AT %MX25236.15 : BOOL;
	bArm1VertStn9Regular_16 AT %MX25236.16 : BOOL;
	bArm1VertStn9Regular_17 AT %MX25236.17 : BOOL;
	bArm1VertStn9Regular_18 AT %MX25236.18 : BOOL;
	bArm1VertStn9Regular_19 AT %MX25236.19 : BOOL;
	bArm1VertStn9Regular_20 AT %MX25236.20 : BOOL;
	bArm1VertStn9Regular_21 AT %MX25236.21 : BOOL;
	bArm1VertStn9Regular_22 AT %MX25236.22 : BOOL;
	bArm1VertStn9Regular_23 AT %MX25236.23 : BOOL;
	bArm1VertStn9Regular_24 AT %MX25236.24 : BOOL;
	bArm1VertStn9Regular_25 AT %MX25236.25 : BOOL;
	bArm1VertStn9Regular_26 AT %MX25236.26 : BOOL;
	bArm1VertStn9Regular_27 AT %MX25236.27 : BOOL;
	bArm1VertStn9Regular_28 AT %MX25236.28 : BOOL;
	bArm1VertStn9Regular_29 AT %MX25236.29 : BOOL;
	bArm1VertStn9Regular_30 AT %MX25236.30 : BOOL;
	bArm1VertStn9Regular_31 AT %MX25236.31 : BOOL;

	bArm1VertStn10Regular_00 AT %MX25240.0 : BOOL;
	bArm1VertStn10Regular_01 AT %MX25240.1 : BOOL;
	bArm1VertStn10Regular_02 AT %MX25240.2 : BOOL;
	bArm1VertStn10Regular_03 AT %MX25240.3 : BOOL;
	bArm1VertStn10Regular_04 AT %MX25240.4 : BOOL;
	bArm1VertStn10Regular_05 AT %MX25240.5 : BOOL;
	bArm1VertStn10Regular_06 AT %MX25240.6 : BOOL;
	bArm1VertStn10Regular_07 AT %MX25240.7 : BOOL;
	bArm1VertStn10Regular_08 AT %MX25240.8 : BOOL;
	bArm1VertStn10Regular_09 AT %MX25240.9 : BOOL;
	bArm1VertStn10Regular_10 AT %MX25240.10 : BOOL;
	bArm1VertStn10Regular_11 AT %MX25240.11 : BOOL;
	bArm1VertStn10Regular_12 AT %MX25240.12 : BOOL;
	bArm1VertStn10Regular_13 AT %MX25240.13 : BOOL;
	bArm1VertStn10Regular_14 AT %MX25240.14 : BOOL;
	bArm1VertStn10Regular_15 AT %MX25240.15 : BOOL;
	bArm1VertStn10Regular_16 AT %MX25240.16 : BOOL;
	bArm1VertStn10Regular_17 AT %MX25240.17 : BOOL;
	bArm1VertStn10Regular_18 AT %MX25240.18 : BOOL;
	bArm1VertStn10Regular_19 AT %MX25240.19 : BOOL;
	bArm1VertStn10Regular_20 AT %MX25240.20 : BOOL;
	bArm1VertStn10Regular_21 AT %MX25240.21 : BOOL;
	bArm1VertStn10Regular_22 AT %MX25240.22 : BOOL;
	bArm1VertStn10Regular_23 AT %MX25240.23 : BOOL;
	bArm1VertStn10Regular_24 AT %MX25240.24 : BOOL;
	bArm1VertStn10Regular_25 AT %MX25240.25 : BOOL;
	bArm1VertStn10Regular_26 AT %MX25240.26 : BOOL;
	bArm1VertStn10Regular_27 AT %MX25240.27 : BOOL;
	bArm1VertStn10Regular_28 AT %MX25240.28 : BOOL;
	bArm1VertStn10Regular_29 AT %MX25240.29 : BOOL;
	bArm1VertStn10Regular_30 AT %MX25240.30 : BOOL;
	bArm1VertStn10Regular_31 AT %MX25240.31 : BOOL;

	bArm1VertStn11Regular_00 AT %MX25244.0 : BOOL;
	bArm1VertStn11Regular_01 AT %MX25244.1 : BOOL;
	bArm1VertStn11Regular_02 AT %MX25244.2 : BOOL;
	bArm1VertStn11Regular_03 AT %MX25244.3 : BOOL;
	bArm1VertStn11Regular_04 AT %MX25244.4 : BOOL;
	bArm1VertStn11Regular_05 AT %MX25244.5 : BOOL;
	bArm1VertStn11Regular_06 AT %MX25244.6 : BOOL;
	bArm1VertStn11Regular_07 AT %MX25244.7 : BOOL;
	bArm1VertStn11Regular_08 AT %MX25244.8 : BOOL;
	bArm1VertStn11Regular_09 AT %MX25244.9 : BOOL;
	bArm1VertStn11Regular_10 AT %MX25244.10 : BOOL;
	bArm1VertStn11Regular_11 AT %MX25244.11 : BOOL;
	bArm1VertStn11Regular_12 AT %MX25244.12 : BOOL;
	bArm1VertStn11Regular_13 AT %MX25244.13 : BOOL;
	bArm1VertStn11Regular_14 AT %MX25244.14 : BOOL;
	bArm1VertStn11Regular_15 AT %MX25244.15 : BOOL;
	bArm1VertStn11Regular_16 AT %MX25244.16 : BOOL;
	bArm1VertStn11Regular_17 AT %MX25244.17 : BOOL;
	bArm1VertStn11Regular_18 AT %MX25244.18 : BOOL;
	bArm1VertStn11Regular_19 AT %MX25244.19 : BOOL;
	bArm1VertStn11Regular_20 AT %MX25244.20 : BOOL;
	bArm1VertStn11Regular_21 AT %MX25244.21 : BOOL;
	bArm1VertStn11Regular_22 AT %MX25244.22 : BOOL;
	bArm1VertStn11Regular_23 AT %MX25244.23 : BOOL;
	bArm1VertStn11Regular_24 AT %MX25244.24 : BOOL;
	bArm1VertStn11Regular_25 AT %MX25244.25 : BOOL;
	bArm1VertStn11Regular_26 AT %MX25244.26 : BOOL;
	bArm1VertStn11Regular_27 AT %MX25244.27 : BOOL;
	bArm1VertStn11Regular_28 AT %MX25244.28 : BOOL;
	bArm1VertStn11Regular_29 AT %MX25244.29 : BOOL;
	bArm1VertStn11Regular_30 AT %MX25244.30 : BOOL;
	bArm1VertStn11Regular_31 AT %MX25244.31 : BOOL;

	bArm1VertStn12Regular_00 AT %MX25248.0 : BOOL;
	bArm1VertStn12Regular_01 AT %MX25248.1 : BOOL;
	bArm1VertStn12Regular_02 AT %MX25248.2 : BOOL;
	bArm1VertStn12Regular_03 AT %MX25248.3 : BOOL;
	bArm1VertStn12Regular_04 AT %MX25248.4 : BOOL;
	bArm1VertStn12Regular_05 AT %MX25248.5 : BOOL;
	bArm1VertStn12Regular_06 AT %MX25248.6 : BOOL;
	bArm1VertStn12Regular_07 AT %MX25248.7 : BOOL;
	bArm1VertStn12Regular_08 AT %MX25248.8 : BOOL;
	bArm1VertStn12Regular_09 AT %MX25248.9 : BOOL;
	bArm1VertStn12Regular_10 AT %MX25248.10 : BOOL;
	bArm1VertStn12Regular_11 AT %MX25248.11 : BOOL;
	bArm1VertStn12Regular_12 AT %MX25248.12 : BOOL;
	bArm1VertStn12Regular_13 AT %MX25248.13 : BOOL;
	bArm1VertStn12Regular_14 AT %MX25248.14 : BOOL;
	bArm1VertStn12Regular_15 AT %MX25248.15 : BOOL;
	bArm1VertStn12Regular_16 AT %MX25248.16 : BOOL;
	bArm1VertStn12Regular_17 AT %MX25248.17 : BOOL;
	bArm1VertStn12Regular_18 AT %MX25248.18 : BOOL;
	bArm1VertStn12Regular_19 AT %MX25248.19 : BOOL;
	bArm1VertStn12Regular_20 AT %MX25248.20 : BOOL;
	bArm1VertStn12Regular_21 AT %MX25248.21 : BOOL;
	bArm1VertStn12Regular_22 AT %MX25248.22 : BOOL;
	bArm1VertStn12Regular_23 AT %MX25248.23 : BOOL;
	bArm1VertStn12Regular_24 AT %MX25248.24 : BOOL;
	bArm1VertStn12Regular_25 AT %MX25248.25 : BOOL;
	bArm1VertStn12Regular_26 AT %MX25248.26 : BOOL;
	bArm1VertStn12Regular_27 AT %MX25248.27 : BOOL;
	bArm1VertStn12Regular_28 AT %MX25248.28 : BOOL;
	bArm1VertStn12Regular_29 AT %MX25248.29 : BOOL;
	bArm1VertStn12Regular_30 AT %MX25248.30 : BOOL;
	bArm1VertStn12Regular_31 AT %MX25248.31 : BOOL;


(* xxxxxxxxxxxxxxxxxxxxxxxxxxxxxxxxxxxxxxx Vert xxxxxxxxxxxxxxxxxxxxxxxxxxxxxxxxxxxxxxx*)
(*========= Up AgiUp BOOL LINK with %MX25300-MX25399 =========*)

	bArm1VertStn1AglUp_00 AT %MX25304.0 : BOOL;
	bArm1VertStn1AglUp_01 AT %MX25304.1 : BOOL;
	bArm1VertStn1AglUp_02 AT %MX25304.2 : BOOL;
	bArm1VertStn1AglUp_03 AT %MX25304.3 : BOOL;
	bArm1VertStn1AglUp_04 AT %MX25304.4 : BOOL;
	bArm1VertStn1AglUp_05 AT %MX25304.5 : BOOL;
	bArm1VertStn1AglUp_06 AT %MX25304.6 : BOOL;
	bArm1VertStn1AglUp_07 AT %MX25304.7 : BOOL;
	bArm1VertStn1AglUp_08 AT %MX25304.8 : BOOL;
	bArm1VertStn1AglUp_09 AT %MX25304.9 : BOOL;
	bArm1VertStn1AglUp_10 AT %MX25304.10 : BOOL;
	bArm1VertStn1AglUp_11 AT %MX25304.11 : BOOL;
	bArm1VertStn1AglUp_12 AT %MX25304.12 : BOOL;
	bArm1VertStn1AglUp_13 AT %MX25304.13 : BOOL;
	bArm1VertStn1AglUp_14 AT %MX25304.14 : BOOL;
	bArm1VertStn1AglUp_15 AT %MX25304.15 : BOOL;
	bArm1VertStn1AglUp_16 AT %MX25304.16 : BOOL;
	bArm1VertStn1AglUp_17 AT %MX25304.17 : BOOL;
	bArm1VertStn1AglUp_18 AT %MX25304.18 : BOOL;
	bArm1VertStn1AglUp_19 AT %MX25304.19 : BOOL;
	bArm1VertStn1AglUp_20 AT %MX25304.20 : BOOL;
	bArm1VertStn1AglUp_21 AT %MX25304.21 : BOOL;
	bArm1VertStn1AglUp_22 AT %MX25304.22 : BOOL;
	bArm1VertStn1AglUp_23 AT %MX25304.23 : BOOL;
	bArm1VertStn1AglUp_24 AT %MX25304.24 : BOOL;
	bArm1VertStn1AglUp_25 AT %MX25304.25 : BOOL;
	bArm1VertStn1AglUp_26 AT %MX25304.26 : BOOL;
	bArm1VertStn1AglUp_27 AT %MX25304.27 : BOOL;
	bArm1VertStn1AglUp_28 AT %MX25304.28 : BOOL;
	bArm1VertStn1AglUp_29 AT %MX25304.29 : BOOL;
	bArm1VertStn1AglUp_30 AT %MX25304.30 : BOOL;
	bArm1VertStn1AglUp_31 AT %MX25304.31 : BOOL;

	bArm1VertStn2AglUp_00 AT %MX25308.0 : BOOL;
	bArm1VertStn2AglUp_01 AT %MX25308.1 : BOOL;
	bArm1VertStn2AglUp_02 AT %MX25308.2 : BOOL;
	bArm1VertStn2AglUp_03 AT %MX25308.3 : BOOL;
	bArm1VertStn2AglUp_04 AT %MX25308.4 : BOOL;
	bArm1VertStn2AglUp_05 AT %MX25308.5 : BOOL;
	bArm1VertStn2AglUp_06 AT %MX25308.6 : BOOL;
	bArm1VertStn2AglUp_07 AT %MX25308.7 : BOOL;
	bArm1VertStn2AglUp_08 AT %MX25308.8 : BOOL;
	bArm1VertStn2AglUp_09 AT %MX25308.9 : BOOL;
	bArm1VertStn2AglUp_10 AT %MX25308.10 : BOOL;
	bArm1VertStn2AglUp_11 AT %MX25308.11 : BOOL;
	bArm1VertStn2AglUp_12 AT %MX25308.12 : BOOL;
	bArm1VertStn2AglUp_13 AT %MX25308.13 : BOOL;
	bArm1VertStn2AglUp_14 AT %MX25308.14 : BOOL;
	bArm1VertStn2AglUp_15 AT %MX25308.15 : BOOL;
	bArm1VertStn2AglUp_16 AT %MX25308.16 : BOOL;
	bArm1VertStn2AglUp_17 AT %MX25308.17 : BOOL;
	bArm1VertStn2AglUp_18 AT %MX25308.18 : BOOL;
	bArm1VertStn2AglUp_19 AT %MX25308.19 : BOOL;
	bArm1VertStn2AglUp_20 AT %MX25308.20 : BOOL;
	bArm1VertStn2AglUp_21 AT %MX25308.21 : BOOL;
	bArm1VertStn2AglUp_22 AT %MX25308.22 : BOOL;
	bArm1VertStn2AglUp_23 AT %MX25308.23 : BOOL;
	bArm1VertStn2AglUp_24 AT %MX25308.24 : BOOL;
	bArm1VertStn2AglUp_25 AT %MX25308.25 : BOOL;
	bArm1VertStn2AglUp_26 AT %MX25308.26 : BOOL;
	bArm1VertStn2AglUp_27 AT %MX25308.27 : BOOL;
	bArm1VertStn2AglUp_28 AT %MX25308.28 : BOOL;
	bArm1VertStn2AglUp_29 AT %MX25308.29 : BOOL;
	bArm1VertStn2AglUp_30 AT %MX25308.30 : BOOL;
	bArm1VertStn2AglUp_31 AT %MX25308.31 : BOOL;

	bArm1VertStn3AglUp_00 AT %MX25312.0 : BOOL;
	bArm1VertStn3AglUp_01 AT %MX25312.1 : BOOL;
	bArm1VertStn3AglUp_02 AT %MX25312.2 : BOOL;
	bArm1VertStn3AglUp_03 AT %MX25312.3 : BOOL;
	bArm1VertStn3AglUp_04 AT %MX25312.4 : BOOL;
	bArm1VertStn3AglUp_05 AT %MX25312.5 : BOOL;
	bArm1VertStn3AglUp_06 AT %MX25312.6 : BOOL;
	bArm1VertStn3AglUp_07 AT %MX25312.7 : BOOL;
	bArm1VertStn3AglUp_08 AT %MX25312.8 : BOOL;
	bArm1VertStn3AglUp_09 AT %MX25312.9 : BOOL;
	bArm1VertStn3AglUp_10 AT %MX25312.10 : BOOL;
	bArm1VertStn3AglUp_11 AT %MX25312.11 : BOOL;
	bArm1VertStn3AglUp_12 AT %MX25312.12 : BOOL;
	bArm1VertStn3AglUp_13 AT %MX25312.13 : BOOL;
	bArm1VertStn3AglUp_14 AT %MX25312.14 : BOOL;
	bArm1VertStn3AglUp_15 AT %MX25312.15 : BOOL;
	bArm1VertStn3AglUp_16 AT %MX25312.16 : BOOL;
	bArm1VertStn3AglUp_17 AT %MX25312.17 : BOOL;
	bArm1VertStn3AglUp_18 AT %MX25312.18 : BOOL;
	bArm1VertStn3AglUp_19 AT %MX25312.19 : BOOL;
	bArm1VertStn3AglUp_20 AT %MX25312.20 : BOOL;
	bArm1VertStn3AglUp_21 AT %MX25312.21 : BOOL;
	bArm1VertStn3AglUp_22 AT %MX25312.22 : BOOL;
	bArm1VertStn3AglUp_23 AT %MX25312.23 : BOOL;
	bArm1VertStn3AglUp_24 AT %MX25312.24 : BOOL;
	bArm1VertStn3AglUp_25 AT %MX25312.25 : BOOL;
	bArm1VertStn3AglUp_26 AT %MX25312.26 : BOOL;
	bArm1VertStn3AglUp_27 AT %MX25312.27 : BOOL;
	bArm1VertStn3AglUp_28 AT %MX25312.28 : BOOL;
	bArm1VertStn3AglUp_29 AT %MX25312.29 : BOOL;
	bArm1VertStn3AglUp_30 AT %MX25312.30 : BOOL;
	bArm1VertStn3AglUp_31 AT %MX25312.31 : BOOL;

	bArm1VertStn4AglUp_00 AT %MX25316.0 : BOOL;
	bArm1VertStn4AglUp_01 AT %MX25316.1 : BOOL;
	bArm1VertStn4AglUp_02 AT %MX25316.2 : BOOL;
	bArm1VertStn4AglUp_03 AT %MX25316.3 : BOOL;
	bArm1VertStn4AglUp_04 AT %MX25316.4 : BOOL;
	bArm1VertStn4AglUp_05 AT %MX25316.5 : BOOL;
	bArm1VertStn4AglUp_06 AT %MX25316.6 : BOOL;
	bArm1VertStn4AglUp_07 AT %MX25316.7 : BOOL;
	bArm1VertStn4AglUp_08 AT %MX25316.8 : BOOL;
	bArm1VertStn4AglUp_09 AT %MX25316.9 : BOOL;
	bArm1VertStn4AglUp_10 AT %MX25316.10 : BOOL;
	bArm1VertStn4AglUp_11 AT %MX25316.11 : BOOL;
	bArm1VertStn4AglUp_12 AT %MX25316.12 : BOOL;
	bArm1VertStn4AglUp_13 AT %MX25316.13 : BOOL;
	bArm1VertStn4AglUp_14 AT %MX25316.14 : BOOL;
	bArm1VertStn4AglUp_15 AT %MX25316.15 : BOOL;
	bArm1VertStn4AglUp_16 AT %MX25316.16 : BOOL;
	bArm1VertStn4AglUp_17 AT %MX25316.17 : BOOL;
	bArm1VertStn4AglUp_18 AT %MX25316.18 : BOOL;
	bArm1VertStn4AglUp_19 AT %MX25316.19 : BOOL;
	bArm1VertStn4AglUp_20 AT %MX25316.20 : BOOL;
	bArm1VertStn4AglUp_21 AT %MX25316.21 : BOOL;
	bArm1VertStn4AglUp_22 AT %MX25316.22 : BOOL;
	bArm1VertStn4AglUp_23 AT %MX25316.23 : BOOL;
	bArm1VertStn4AglUp_24 AT %MX25316.24 : BOOL;
	bArm1VertStn4AglUp_25 AT %MX25316.25 : BOOL;
	bArm1VertStn4AglUp_26 AT %MX25316.26 : BOOL;
	bArm1VertStn4AglUp_27 AT %MX25316.27 : BOOL;
	bArm1VertStn4AglUp_28 AT %MX25316.28 : BOOL;
	bArm1VertStn4AglUp_29 AT %MX25316.29 : BOOL;
	bArm1VertStn4AglUp_30 AT %MX25316.30 : BOOL;
	bArm1VertStn4AglUp_31 AT %MX25316.31 : BOOL;

	bArm1VertStn5AglUp_00 AT %MX25320.0 : BOOL;
	bArm1VertStn5AglUp_01 AT %MX25320.1 : BOOL;
	bArm1VertStn5AglUp_02 AT %MX25320.2 : BOOL;
	bArm1VertStn5AglUp_03 AT %MX25320.3 : BOOL;
	bArm1VertStn5AglUp_04 AT %MX25320.4 : BOOL;
	bArm1VertStn5AglUp_05 AT %MX25320.5 : BOOL;
	bArm1VertStn5AglUp_06 AT %MX25320.6 : BOOL;
	bArm1VertStn5AglUp_07 AT %MX25320.7 : BOOL;
	bArm1VertStn5AglUp_08 AT %MX25320.8 : BOOL;
	bArm1VertStn5AglUp_09 AT %MX25320.9 : BOOL;
	bArm1VertStn5AglUp_10 AT %MX25320.10 : BOOL;
	bArm1VertStn5AglUp_11 AT %MX25320.11 : BOOL;
	bArm1VertStn5AglUp_12 AT %MX25320.12 : BOOL;
	bArm1VertStn5AglUp_13 AT %MX25320.13 : BOOL;
	bArm1VertStn5AglUp_14 AT %MX25320.14 : BOOL;
	bArm1VertStn5AglUp_15 AT %MX25320.15 : BOOL;
	bArm1VertStn5AglUp_16 AT %MX25320.16 : BOOL;
	bArm1VertStn5AglUp_17 AT %MX25320.17 : BOOL;
	bArm1VertStn5AglUp_18 AT %MX25320.18 : BOOL;
	bArm1VertStn5AglUp_19 AT %MX25320.19 : BOOL;
	bArm1VertStn5AglUp_20 AT %MX25320.20 : BOOL;
	bArm1VertStn5AglUp_21 AT %MX25320.21 : BOOL;
	bArm1VertStn5AglUp_22 AT %MX25320.22 : BOOL;
	bArm1VertStn5AglUp_23 AT %MX25320.23 : BOOL;
	bArm1VertStn5AglUp_24 AT %MX25320.24 : BOOL;
	bArm1VertStn5AglUp_25 AT %MX25320.25 : BOOL;
	bArm1VertStn5AglUp_26 AT %MX25320.26 : BOOL;
	bArm1VertStn5AglUp_27 AT %MX25320.27 : BOOL;
	bArm1VertStn5AglUp_28 AT %MX25320.28 : BOOL;
	bArm1VertStn5AglUp_29 AT %MX25320.29 : BOOL;
	bArm1VertStn5AglUp_30 AT %MX25320.30 : BOOL;
	bArm1VertStn5AglUp_31 AT %MX25320.31 : BOOL;

	bArm1VertStn6AglUp_00 AT %MX25324.0 : BOOL;
	bArm1VertStn6AglUp_01 AT %MX25324.1 : BOOL;
	bArm1VertStn6AglUp_02 AT %MX25324.2 : BOOL;
	bArm1VertStn6AglUp_03 AT %MX25324.3 : BOOL;
	bArm1VertStn6AglUp_04 AT %MX25324.4 : BOOL;
	bArm1VertStn6AglUp_05 AT %MX25324.5 : BOOL;
	bArm1VertStn6AglUp_06 AT %MX25324.6 : BOOL;
	bArm1VertStn6AglUp_07 AT %MX25324.7 : BOOL;
	bArm1VertStn6AglUp_08 AT %MX25324.8 : BOOL;
	bArm1VertStn6AglUp_09 AT %MX25324.9 : BOOL;
	bArm1VertStn6AglUp_10 AT %MX25324.10 : BOOL;
	bArm1VertStn6AglUp_11 AT %MX25324.11 : BOOL;
	bArm1VertStn6AglUp_12 AT %MX25324.12 : BOOL;
	bArm1VertStn6AglUp_13 AT %MX25324.13 : BOOL;
	bArm1VertStn6AglUp_14 AT %MX25324.14 : BOOL;
	bArm1VertStn6AglUp_15 AT %MX25324.15 : BOOL;
	bArm1VertStn6AglUp_16 AT %MX25324.16 : BOOL;
	bArm1VertStn6AglUp_17 AT %MX25324.17 : BOOL;
	bArm1VertStn6AglUp_18 AT %MX25324.18 : BOOL;
	bArm1VertStn6AglUp_19 AT %MX25324.19 : BOOL;
	bArm1VertStn6AglUp_20 AT %MX25324.20 : BOOL;
	bArm1VertStn6AglUp_21 AT %MX25324.21 : BOOL;
	bArm1VertStn6AglUp_22 AT %MX25324.22 : BOOL;
	bArm1VertStn6AglUp_23 AT %MX25324.23 : BOOL;
	bArm1VertStn6AglUp_24 AT %MX25324.24 : BOOL;
	bArm1VertStn6AglUp_25 AT %MX25324.25 : BOOL;
	bArm1VertStn6AglUp_26 AT %MX25324.26 : BOOL;
	bArm1VertStn6AglUp_27 AT %MX25324.27 : BOOL;
	bArm1VertStn6AglUp_28 AT %MX25324.28 : BOOL;
	bArm1VertStn6AglUp_29 AT %MX25324.29 : BOOL;
	bArm1VertStn6AglUp_30 AT %MX25324.30 : BOOL;
	bArm1VertStn6AglUp_31 AT %MX25324.31 : BOOL;

	bArm1VertStn7AglUp_00 AT %MX25328.0 : BOOL;
	bArm1VertStn7AglUp_01 AT %MX25328.1 : BOOL;
	bArm1VertStn7AglUp_02 AT %MX25328.2 : BOOL;
	bArm1VertStn7AglUp_03 AT %MX25328.3 : BOOL;
	bArm1VertStn7AglUp_04 AT %MX25328.4 : BOOL;
	bArm1VertStn7AglUp_05 AT %MX25328.5 : BOOL;
	bArm1VertStn7AglUp_06 AT %MX25328.6 : BOOL;
	bArm1VertStn7AglUp_07 AT %MX25328.7 : BOOL;
	bArm1VertStn7AglUp_08 AT %MX25328.8 : BOOL;
	bArm1VertStn7AglUp_09 AT %MX25328.9 : BOOL;
	bArm1VertStn7AglUp_10 AT %MX25328.10 : BOOL;
	bArm1VertStn7AglUp_11 AT %MX25328.11 : BOOL;
	bArm1VertStn7AglUp_12 AT %MX25328.12 : BOOL;
	bArm1VertStn7AglUp_13 AT %MX25328.13 : BOOL;
	bArm1VertStn7AglUp_14 AT %MX25328.14 : BOOL;
	bArm1VertStn7AglUp_15 AT %MX25328.15 : BOOL;
	bArm1VertStn7AglUp_16 AT %MX25328.16 : BOOL;
	bArm1VertStn7AglUp_17 AT %MX25328.17 : BOOL;
	bArm1VertStn7AglUp_18 AT %MX25328.18 : BOOL;
	bArm1VertStn7AglUp_19 AT %MX25328.19 : BOOL;
	bArm1VertStn7AglUp_20 AT %MX25328.20 : BOOL;
	bArm1VertStn7AglUp_21 AT %MX25328.21 : BOOL;
	bArm1VertStn7AglUp_22 AT %MX25328.22 : BOOL;
	bArm1VertStn7AglUp_23 AT %MX25328.23 : BOOL;
	bArm1VertStn7AglUp_24 AT %MX25328.24 : BOOL;
	bArm1VertStn7AglUp_25 AT %MX25328.25 : BOOL;
	bArm1VertStn7AglUp_26 AT %MX25328.26 : BOOL;
	bArm1VertStn7AglUp_27 AT %MX25328.27 : BOOL;
	bArm1VertStn7AglUp_28 AT %MX25328.28 : BOOL;
	bArm1VertStn7AglUp_29 AT %MX25328.29 : BOOL;
	bArm1VertStn7AglUp_30 AT %MX25328.30 : BOOL;
	bArm1VertStn7AglUp_31 AT %MX25328.31 : BOOL;

	bArm1VertStn8AglUp_00 AT %MX25332.0 : BOOL;
	bArm1VertStn8AglUp_01 AT %MX25332.1 : BOOL;
	bArm1VertStn8AglUp_02 AT %MX25332.2 : BOOL;
	bArm1VertStn8AglUp_03 AT %MX25332.3 : BOOL;
	bArm1VertStn8AglUp_04 AT %MX25332.4 : BOOL;
	bArm1VertStn8AglUp_05 AT %MX25332.5 : BOOL;
	bArm1VertStn8AglUp_06 AT %MX25332.6 : BOOL;
	bArm1VertStn8AglUp_07 AT %MX25332.7 : BOOL;
	bArm1VertStn8AglUp_08 AT %MX25332.8 : BOOL;
	bArm1VertStn8AglUp_09 AT %MX25332.9 : BOOL;
	bArm1VertStn8AglUp_10 AT %MX25332.10 : BOOL;
	bArm1VertStn8AglUp_11 AT %MX25332.11 : BOOL;
	bArm1VertStn8AglUp_12 AT %MX25332.12 : BOOL;
	bArm1VertStn8AglUp_13 AT %MX25332.13 : BOOL;
	bArm1VertStn8AglUp_14 AT %MX25332.14 : BOOL;
	bArm1VertStn8AglUp_15 AT %MX25332.15 : BOOL;
	bArm1VertStn8AglUp_16 AT %MX25332.16 : BOOL;
	bArm1VertStn8AglUp_17 AT %MX25332.17 : BOOL;
	bArm1VertStn8AglUp_18 AT %MX25332.18 : BOOL;
	bArm1VertStn8AglUp_19 AT %MX25332.19 : BOOL;
	bArm1VertStn8AglUp_20 AT %MX25332.20 : BOOL;
	bArm1VertStn8AglUp_21 AT %MX25332.21 : BOOL;
	bArm1VertStn8AglUp_22 AT %MX25332.22 : BOOL;
	bArm1VertStn8AglUp_23 AT %MX25332.23 : BOOL;
	bArm1VertStn8AglUp_24 AT %MX25332.24 : BOOL;
	bArm1VertStn8AglUp_25 AT %MX25332.25 : BOOL;
	bArm1VertStn8AglUp_26 AT %MX25332.26 : BOOL;
	bArm1VertStn8AglUp_27 AT %MX25332.27 : BOOL;
	bArm1VertStn8AglUp_28 AT %MX25332.28 : BOOL;
	bArm1VertStn8AglUp_29 AT %MX25332.29 : BOOL;
	bArm1VertStn8AglUp_30 AT %MX25332.30 : BOOL;
	bArm1VertStn8AglUp_31 AT %MX25332.31 : BOOL;

	bArm1VertStn9AglUp_00 AT %MX25336.0 : BOOL;
	bArm1VertStn9AglUp_01 AT %MX25336.1 : BOOL;
	bArm1VertStn9AglUp_02 AT %MX25336.2 : BOOL;
	bArm1VertStn9AglUp_03 AT %MX25336.3 : BOOL;
	bArm1VertStn9AglUp_04 AT %MX25336.4 : BOOL;
	bArm1VertStn9AglUp_05 AT %MX25336.5 : BOOL;
	bArm1VertStn9AglUp_06 AT %MX25336.6 : BOOL;
	bArm1VertStn9AglUp_07 AT %MX25336.7 : BOOL;
	bArm1VertStn9AglUp_08 AT %MX25336.8 : BOOL;
	bArm1VertStn9AglUp_09 AT %MX25336.9 : BOOL;
	bArm1VertStn9AglUp_10 AT %MX25336.10 : BOOL;
	bArm1VertStn9AglUp_11 AT %MX25336.11 : BOOL;
	bArm1VertStn9AglUp_12 AT %MX25336.12 : BOOL;
	bArm1VertStn9AglUp_13 AT %MX25336.13 : BOOL;
	bArm1VertStn9AglUp_14 AT %MX25336.14 : BOOL;
	bArm1VertStn9AglUp_15 AT %MX25336.15 : BOOL;
	bArm1VertStn9AglUp_16 AT %MX25336.16 : BOOL;
	bArm1VertStn9AglUp_17 AT %MX25336.17 : BOOL;
	bArm1VertStn9AglUp_18 AT %MX25336.18 : BOOL;
	bArm1VertStn9AglUp_19 AT %MX25336.19 : BOOL;
	bArm1VertStn9AglUp_20 AT %MX25336.20 : BOOL;
	bArm1VertStn9AglUp_21 AT %MX25336.21 : BOOL;
	bArm1VertStn9AglUp_22 AT %MX25336.22 : BOOL;
	bArm1VertStn9AglUp_23 AT %MX25336.23 : BOOL;
	bArm1VertStn9AglUp_24 AT %MX25336.24 : BOOL;
	bArm1VertStn9AglUp_25 AT %MX25336.25 : BOOL;
	bArm1VertStn9AglUp_26 AT %MX25336.26 : BOOL;
	bArm1VertStn9AglUp_27 AT %MX25336.27 : BOOL;
	bArm1VertStn9AglUp_28 AT %MX25336.28 : BOOL;
	bArm1VertStn9AglUp_29 AT %MX25336.29 : BOOL;
	bArm1VertStn9AglUp_30 AT %MX25336.30 : BOOL;
	bArm1VertStn9AglUp_31 AT %MX25336.31 : BOOL;

	bArm1VertStn10AglUp_00 AT %MX25340.0 : BOOL;
	bArm1VertStn10AglUp_01 AT %MX25340.1 : BOOL;
	bArm1VertStn10AglUp_02 AT %MX25340.2 : BOOL;
	bArm1VertStn10AglUp_03 AT %MX25340.3 : BOOL;
	bArm1VertStn10AglUp_04 AT %MX25340.4 : BOOL;
	bArm1VertStn10AglUp_05 AT %MX25340.5 : BOOL;
	bArm1VertStn10AglUp_06 AT %MX25340.6 : BOOL;
	bArm1VertStn10AglUp_07 AT %MX25340.7 : BOOL;
	bArm1VertStn10AglUp_08 AT %MX25340.8 : BOOL;
	bArm1VertStn10AglUp_09 AT %MX25340.9 : BOOL;
	bArm1VertStn10AglUp_10 AT %MX25340.10 : BOOL;
	bArm1VertStn10AglUp_11 AT %MX25340.11 : BOOL;
	bArm1VertStn10AglUp_12 AT %MX25340.12 : BOOL;
	bArm1VertStn10AglUp_13 AT %MX25340.13 : BOOL;
	bArm1VertStn10AglUp_14 AT %MX25340.14 : BOOL;
	bArm1VertStn10AglUp_15 AT %MX25340.15 : BOOL;
	bArm1VertStn10AglUp_16 AT %MX25340.16 : BOOL;
	bArm1VertStn10AglUp_17 AT %MX25340.17 : BOOL;
	bArm1VertStn10AglUp_18 AT %MX25340.18 : BOOL;
	bArm1VertStn10AglUp_19 AT %MX25340.19 : BOOL;
	bArm1VertStn10AglUp_20 AT %MX25340.20 : BOOL;
	bArm1VertStn10AglUp_21 AT %MX25340.21 : BOOL;
	bArm1VertStn10AglUp_22 AT %MX25340.22 : BOOL;
	bArm1VertStn10AglUp_23 AT %MX25340.23 : BOOL;
	bArm1VertStn10AglUp_24 AT %MX25340.24 : BOOL;
	bArm1VertStn10AglUp_25 AT %MX25340.25 : BOOL;
	bArm1VertStn10AglUp_26 AT %MX25340.26 : BOOL;
	bArm1VertStn10AglUp_27 AT %MX25340.27 : BOOL;
	bArm1VertStn10AglUp_28 AT %MX25340.28 : BOOL;
	bArm1VertStn10AglUp_29 AT %MX25340.29 : BOOL;
	bArm1VertStn10AglUp_30 AT %MX25340.30 : BOOL;
	bArm1VertStn10AglUp_31 AT %MX25340.31 : BOOL;

	bArm1VertStn11AglUp_00 AT %MX25344.0 : BOOL;
	bArm1VertStn11AglUp_01 AT %MX25344.1 : BOOL;
	bArm1VertStn11AglUp_02 AT %MX25344.2 : BOOL;
	bArm1VertStn11AglUp_03 AT %MX25344.3 : BOOL;
	bArm1VertStn11AglUp_04 AT %MX25344.4 : BOOL;
	bArm1VertStn11AglUp_05 AT %MX25344.5 : BOOL;
	bArm1VertStn11AglUp_06 AT %MX25344.6 : BOOL;
	bArm1VertStn11AglUp_07 AT %MX25344.7 : BOOL;
	bArm1VertStn11AglUp_08 AT %MX25344.8 : BOOL;
	bArm1VertStn11AglUp_09 AT %MX25344.9 : BOOL;
	bArm1VertStn11AglUp_10 AT %MX25344.10 : BOOL;
	bArm1VertStn11AglUp_11 AT %MX25344.11 : BOOL;
	bArm1VertStn11AglUp_12 AT %MX25344.12 : BOOL;
	bArm1VertStn11AglUp_13 AT %MX25344.13 : BOOL;
	bArm1VertStn11AglUp_14 AT %MX25344.14 : BOOL;
	bArm1VertStn11AglUp_15 AT %MX25344.15 : BOOL;
	bArm1VertStn11AglUp_16 AT %MX25344.16 : BOOL;
	bArm1VertStn11AglUp_17 AT %MX25344.17 : BOOL;
	bArm1VertStn11AglUp_18 AT %MX25344.18 : BOOL;
	bArm1VertStn11AglUp_19 AT %MX25344.19 : BOOL;
	bArm1VertStn11AglUp_20 AT %MX25344.20 : BOOL;
	bArm1VertStn11AglUp_21 AT %MX25344.21 : BOOL;
	bArm1VertStn11AglUp_22 AT %MX25344.22 : BOOL;
	bArm1VertStn11AglUp_23 AT %MX25344.23 : BOOL;
	bArm1VertStn11AglUp_24 AT %MX25344.24 : BOOL;
	bArm1VertStn11AglUp_25 AT %MX25344.25 : BOOL;
	bArm1VertStn11AglUp_26 AT %MX25344.26 : BOOL;
	bArm1VertStn11AglUp_27 AT %MX25344.27 : BOOL;
	bArm1VertStn11AglUp_28 AT %MX25344.28 : BOOL;
	bArm1VertStn11AglUp_29 AT %MX25344.29 : BOOL;
	bArm1VertStn11AglUp_30 AT %MX25344.30 : BOOL;
	bArm1VertStn11AglUp_31 AT %MX25344.31 : BOOL;

	bArm1VertStn12AglUp_00 AT %MX25348.0 : BOOL;
	bArm1VertStn12AglUp_01 AT %MX25348.1 : BOOL;
	bArm1VertStn12AglUp_02 AT %MX25348.2 : BOOL;
	bArm1VertStn12AglUp_03 AT %MX25348.3 : BOOL;
	bArm1VertStn12AglUp_04 AT %MX25348.4 : BOOL;
	bArm1VertStn12AglUp_05 AT %MX25348.5 : BOOL;
	bArm1VertStn12AglUp_06 AT %MX25348.6 : BOOL;
	bArm1VertStn12AglUp_07 AT %MX25348.7 : BOOL;
	bArm1VertStn12AglUp_08 AT %MX25348.8 : BOOL;
	bArm1VertStn12AglUp_09 AT %MX25348.9 : BOOL;
	bArm1VertStn12AglUp_10 AT %MX25348.10 : BOOL;
	bArm1VertStn12AglUp_11 AT %MX25348.11 : BOOL;
	bArm1VertStn12AglUp_12 AT %MX25348.12 : BOOL;
	bArm1VertStn12AglUp_13 AT %MX25348.13 : BOOL;
	bArm1VertStn12AglUp_14 AT %MX25348.14 : BOOL;
	bArm1VertStn12AglUp_15 AT %MX25348.15 : BOOL;
	bArm1VertStn12AglUp_16 AT %MX25348.16 : BOOL;
	bArm1VertStn12AglUp_17 AT %MX25348.17 : BOOL;
	bArm1VertStn12AglUp_18 AT %MX25348.18 : BOOL;
	bArm1VertStn12AglUp_19 AT %MX25348.19 : BOOL;
	bArm1VertStn12AglUp_20 AT %MX25348.20 : BOOL;
	bArm1VertStn12AglUp_21 AT %MX25348.21 : BOOL;
	bArm1VertStn12AglUp_22 AT %MX25348.22 : BOOL;
	bArm1VertStn12AglUp_23 AT %MX25348.23 : BOOL;
	bArm1VertStn12AglUp_24 AT %MX25348.24 : BOOL;
	bArm1VertStn12AglUp_25 AT %MX25348.25 : BOOL;
	bArm1VertStn12AglUp_26 AT %MX25348.26 : BOOL;
	bArm1VertStn12AglUp_27 AT %MX25348.27 : BOOL;
	bArm1VertStn12AglUp_28 AT %MX25348.28 : BOOL;
	bArm1VertStn12AglUp_29 AT %MX25348.29 : BOOL;
	bArm1VertStn12AglUp_30 AT %MX25348.30 : BOOL;
	bArm1VertStn12AglUp_31 AT %MX25348.31 : BOOL;


(* xxxxxxxxxxxxxxxxxxxxxxxxxxxxxxxxxxxxxxx Vert xxxxxxxxxxxxxxxxxxxxxxxxxxxxxxxxxxxxxxx*)
(*========= Down AgiDown BOOL LINK with %MX25400-MX25499 =========*)

	bArm1VertStn1AglDown_00 AT %MX25404.0 : BOOL;
	bArm1VertStn1AglDown_01 AT %MX25404.1 : BOOL;
	bArm1VertStn1AglDown_02 AT %MX25404.2 : BOOL;
	bArm1VertStn1AglDown_03 AT %MX25404.3 : BOOL;
	bArm1VertStn1AglDown_04 AT %MX25404.4 : BOOL;
	bArm1VertStn1AglDown_05 AT %MX25404.5 : BOOL;
	bArm1VertStn1AglDown_06 AT %MX25404.6 : BOOL;
	bArm1VertStn1AglDown_07 AT %MX25404.7 : BOOL;
	bArm1VertStn1AglDown_08 AT %MX25404.8 : BOOL;
	bArm1VertStn1AglDown_09 AT %MX25404.9 : BOOL;
	bArm1VertStn1AglDown_10 AT %MX25404.10 : BOOL;
	bArm1VertStn1AglDown_11 AT %MX25404.11 : BOOL;
	bArm1VertStn1AglDown_12 AT %MX25404.12 : BOOL;
	bArm1VertStn1AglDown_13 AT %MX25404.13 : BOOL;
	bArm1VertStn1AglDown_14 AT %MX25404.14 : BOOL;
	bArm1VertStn1AglDown_15 AT %MX25404.15 : BOOL;
	bArm1VertStn1AglDown_16 AT %MX25404.16 : BOOL;
	bArm1VertStn1AglDown_17 AT %MX25404.17 : BOOL;
	bArm1VertStn1AglDown_18 AT %MX25404.18 : BOOL;
	bArm1VertStn1AglDown_19 AT %MX25404.19 : BOOL;
	bArm1VertStn1AglDown_20 AT %MX25404.20 : BOOL;
	bArm1VertStn1AglDown_21 AT %MX25404.21 : BOOL;
	bArm1VertStn1AglDown_22 AT %MX25404.22 : BOOL;
	bArm1VertStn1AglDown_23 AT %MX25404.23 : BOOL;
	bArm1VertStn1AglDown_24 AT %MX25404.24 : BOOL;
	bArm1VertStn1AglDown_25 AT %MX25404.25 : BOOL;
	bArm1VertStn1AglDown_26 AT %MX25404.26 : BOOL;
	bArm1VertStn1AglDown_27 AT %MX25404.27 : BOOL;
	bArm1VertStn1AglDown_28 AT %MX25404.28 : BOOL;
	bArm1VertStn1AglDown_29 AT %MX25404.29 : BOOL;
	bArm1VertStn1AglDown_30 AT %MX25404.30 : BOOL;
	bArm1VertStn1AglDown_31 AT %MX25404.31 : BOOL;

	bArm1VertStn2AglDown_00 AT %MX25408.0 : BOOL;
	bArm1VertStn2AglDown_01 AT %MX25408.1 : BOOL;
	bArm1VertStn2AglDown_02 AT %MX25408.2 : BOOL;
	bArm1VertStn2AglDown_03 AT %MX25408.3 : BOOL;
	bArm1VertStn2AglDown_04 AT %MX25408.4 : BOOL;
	bArm1VertStn2AglDown_05 AT %MX25408.5 : BOOL;
	bArm1VertStn2AglDown_06 AT %MX25408.6 : BOOL;
	bArm1VertStn2AglDown_07 AT %MX25408.7 : BOOL;
	bArm1VertStn2AglDown_08 AT %MX25408.8 : BOOL;
	bArm1VertStn2AglDown_09 AT %MX25408.9 : BOOL;
	bArm1VertStn2AglDown_10 AT %MX25408.10 : BOOL;
	bArm1VertStn2AglDown_11 AT %MX25408.11 : BOOL;
	bArm1VertStn2AglDown_12 AT %MX25408.12 : BOOL;
	bArm1VertStn2AglDown_13 AT %MX25408.13 : BOOL;
	bArm1VertStn2AglDown_14 AT %MX25408.14 : BOOL;
	bArm1VertStn2AglDown_15 AT %MX25408.15 : BOOL;
	bArm1VertStn2AglDown_16 AT %MX25408.16 : BOOL;
	bArm1VertStn2AglDown_17 AT %MX25408.17 : BOOL;
	bArm1VertStn2AglDown_18 AT %MX25408.18 : BOOL;
	bArm1VertStn2AglDown_19 AT %MX25408.19 : BOOL;
	bArm1VertStn2AglDown_20 AT %MX25408.20 : BOOL;
	bArm1VertStn2AglDown_21 AT %MX25408.21 : BOOL;
	bArm1VertStn2AglDown_22 AT %MX25408.22 : BOOL;
	bArm1VertStn2AglDown_23 AT %MX25408.23 : BOOL;
	bArm1VertStn2AglDown_24 AT %MX25408.24 : BOOL;
	bArm1VertStn2AglDown_25 AT %MX25408.25 : BOOL;
	bArm1VertStn2AglDown_26 AT %MX25408.26 : BOOL;
	bArm1VertStn2AglDown_27 AT %MX25408.27 : BOOL;
	bArm1VertStn2AglDown_28 AT %MX25408.28 : BOOL;
	bArm1VertStn2AglDown_29 AT %MX25408.29 : BOOL;
	bArm1VertStn2AglDown_30 AT %MX25408.30 : BOOL;
	bArm1VertStn2AglDown_31 AT %MX25408.31 : BOOL;

	bArm1VertStn3AglDown_00 AT %MX25412.0 : BOOL;
	bArm1VertStn3AglDown_01 AT %MX25412.1 : BOOL;
	bArm1VertStn3AglDown_02 AT %MX25412.2 : BOOL;
	bArm1VertStn3AglDown_03 AT %MX25412.3 : BOOL;
	bArm1VertStn3AglDown_04 AT %MX25412.4 : BOOL;
	bArm1VertStn3AglDown_05 AT %MX25412.5 : BOOL;
	bArm1VertStn3AglDown_06 AT %MX25412.6 : BOOL;
	bArm1VertStn3AglDown_07 AT %MX25412.7 : BOOL;
	bArm1VertStn3AglDown_08 AT %MX25412.8 : BOOL;
	bArm1VertStn3AglDown_09 AT %MX25412.9 : BOOL;
	bArm1VertStn3AglDown_10 AT %MX25412.10 : BOOL;
	bArm1VertStn3AglDown_11 AT %MX25412.11 : BOOL;
	bArm1VertStn3AglDown_12 AT %MX25412.12 : BOOL;
	bArm1VertStn3AglDown_13 AT %MX25412.13 : BOOL;
	bArm1VertStn3AglDown_14 AT %MX25412.14 : BOOL;
	bArm1VertStn3AglDown_15 AT %MX25412.15 : BOOL;
	bArm1VertStn3AglDown_16 AT %MX25412.16 : BOOL;
	bArm1VertStn3AglDown_17 AT %MX25412.17 : BOOL;
	bArm1VertStn3AglDown_18 AT %MX25412.18 : BOOL;
	bArm1VertStn3AglDown_19 AT %MX25412.19 : BOOL;
	bArm1VertStn3AglDown_20 AT %MX25412.20 : BOOL;
	bArm1VertStn3AglDown_21 AT %MX25412.21 : BOOL;
	bArm1VertStn3AglDown_22 AT %MX25412.22 : BOOL;
	bArm1VertStn3AglDown_23 AT %MX25412.23 : BOOL;
	bArm1VertStn3AglDown_24 AT %MX25412.24 : BOOL;
	bArm1VertStn3AglDown_25 AT %MX25412.25 : BOOL;
	bArm1VertStn3AglDown_26 AT %MX25412.26 : BOOL;
	bArm1VertStn3AglDown_27 AT %MX25412.27 : BOOL;
	bArm1VertStn3AglDown_28 AT %MX25412.28 : BOOL;
	bArm1VertStn3AglDown_29 AT %MX25412.29 : BOOL;
	bArm1VertStn3AglDown_30 AT %MX25412.30 : BOOL;
	bArm1VertStn3AglDown_31 AT %MX25412.31 : BOOL;

